	ELSE (* command not yet active *)
		IF F_AxisIsCoupled(Axis.NcToPlc.CoupleState) THEN	(* 20090205 KSt *)
			(* if axis is coupled during motion (FlyingSaw) all commands are aborted - 20090205 KSt*)
			CommandAborted := TRUE;
			iState := STATE_INITIALIZATION;
		ELSIF Axis.NcToPlc.CmdNo = 0 AND NcCyclicFeedbackExpected THEN  				(* 20090206 KSt *)
			CounterCmdNoZero := CounterCmdNoZero + 1;
			IF CounterCmdNoZero > TcMcGlobal.NCTOPLC_FEEDBACK_MAXWAITCYCLES THEN (* wait for a certain number of cycles before error *)
				(* CmdNo zero is not supposed to happen - it may come up after a coupling situation for a few cycles *)
				Error := TRUE;
				ErrorID := MC_ERROR_BUFFERED_COMMAND_CMDNOZERO; (* no command state feedback from NC *)
				iState := STATE_INITIALIZATION;
			END_IF
																														(*		ELSIF Axis.NcToPlc.CmdNo = (sStartResponse.nCmdNo + 1) OR
																																     	((Axis.NcToPlc.CmdNo = 1) AND  (sStartResponse.nCmdNo=16#FFFF)) *) 	(* overrun with a difference of 1*) 
		ELSIF DiffCmdNo=1 THEN (* running command number is 1 higher than expected *) (* 20110421 KSt *)
			(* feedback CmdNo is exactly ONE increment higher than my command *)
			(* command was aborted or successfully finished *)
			Error := GETBIT32(Axis.NcToPlc.CmdState, INT_TO_SINT(CMDSTATE_LASTCMD_ENDED_WITH_ERROR));
			CommandAborted := NOT Error AND GETBIT32(Axis.NcToPlc.CmdState, INT_TO_SINT(CMDSTATE_LASTCMD_ABORTED_WITHOUT_ERROR));
(*			Done := NOT Error AND NOT Done AND GETBIT32(Axis.NcToPlc.CmdState, INT_TO_SINT(CMDSTATE_LASTCMD_SUCCESSFULLY_EXECUTED));*)	(* 20100514 KSt *)
			Done := NOT Error AND NOT CommandAborted AND GETBIT32(Axis.NcToPlc.CmdState, INT_TO_SINT(CMDSTATE_LASTCMD_SUCCESSFULLY_EXECUTED));	(* 20100514 KSt *)
			IF Error THEN
				(* if axis error-Id is valid then feed it back - otherwhise errror-Id is unknown. *)
				ErrorID := SEL(Axis.NcToPlc.ErrorCode=0, Axis.NcToPlc.ErrorCode, INT_TO_UDINT(MC_ERROR_BUFFERED_COMMAND_ERRORID_NOT_AVAILABLE) );
			END_IF
			IF NOT Done AND NOT CommandAborted AND NOT Error THEN
				Error := TRUE;
				ErrorID := MC_ERROR_BUFFERED_COMMAND_NO_STATE_FEEDBACK; (* no command state feedback from NC *)
			END_IF
			iState := STATE_INITIALIZATION;
		ELSIF DiffCmdNo=2 THEN (* running command number is 2 higher than expected *) (* 20110421 KSt *)
			(* feedback CmdNo is exactly TWO increments higher than my command  - 20090116 KSt *)
			Error := GETBIT32(Axis.NcToPlc.CmdState, INT_TO_SINT(CMDSTATE_LASTCMD_ENDED_WITH_ERROR)); (* error of command+1 *)
			(* if command+1 was aborted then this command has been aborted as well *)
			CommandAborted := NOT Error AND GETBIT32(Axis.NcToPlc.CmdState, INT_TO_SINT(CMDSTATE_LASTCMD_ABORTED_WITHOUT_ERROR));
			IF NOT CommandAborted THEN
				(* if previous command has not been aborted - the status of this command is unknown *)
				Error := TRUE;	(* command monitoring not possible; probably because function block was not called cyclically *)
				ErrorID := SEL( DiffCycleCounter > 1, INT_TO_UDINT(MC_ERROR_BUFFERED_COMMAND_MONITORING_IMPOSSIBLE), INT_TO_UDINT(MC_ERROR_BUFFCMD_MONITRNGIMPOSS_FBNOTCALLEDCYC));	(* additional error code with command aborted - command monitoring impossible because the block is not called cyclically - 2011-08-01 KSt *)
			END_IF
			iState := STATE_INITIALIZATION;
		ELSIF DiffCmdNo > 0 THEN (* running command number is 3 or more higher than expected *) (* 20110421 KSt *)
			(* feedback CmdNo is THREE or more increments higher than my command *)
			(* command was aborted - command monitoring impossible *)
			Error := TRUE; 	(* command monitoring not possible; probably because function block was not called cyclically *)
			ErrorID := SEL( DiffCycleCounter > 1, INT_TO_UDINT(MC_ERROR_BUFFERED_COMMAND_MONITORING_IMPOSSIBLE), INT_TO_UDINT(MC_ERROR_BUFFCMD_MONITRNGIMPOSS_FBNOTCALLEDCYC)); (* additional error code with command aborted - command monitoring impossible because the block is not called cyclically - 2011-08-01 KSt *)
			(*CommandAborted := TRUE;*)	(*  20090116 KSt *)
			iState := STATE_INITIALIZATION;
		ELSIF F_AxisInErrorState(Axis.NcToPlc.StateDWord) THEN
			(* axis error came up before this command has been started *)
			Error := TRUE;
			ErrorID := AXIS.NcToPlc.ErrorCode;
			iState := STATE_INITIALIZATION;
		ELSIF NOT F_AxisHasJob(Axis.NcToPlc.StateDWord) AND NcCyclicFeedbackExpected THEN
			(* CmdNo is still lower than my command - command has not been initiated *)
			IF F_AxisHasBeenStopped(Axis.NcToPlc.StateDWord) THEN
				CommandAborted := TRUE;		(* stopp command aborts this command *)
				iState := STATE_INITIALIZATION;
			ELSE
				(* other cases are not supposed to happen and are error conditions *)
				CounterCmdNotStarted := CounterCmdNotStarted + 1;
				IF CounterCmdNotStarted > TcMcGlobal.NCTOPLC_FEEDBACK_MAXWAITCYCLES THEN (* wait for a certain number of cycles before error *)
					Error := TRUE;
					ErrorID := MC_ERROR_BUFFERED_COMMAND_NOT_STARTED; (* reason unknown *)
					iState := STATE_INITIALIZATION;
				END_IF
			END_IF
			(* timeout check *);
		END_IF
	END_IF
	IF (Error OR CommandAborted) AND (iState<>STATE_RUNNING) THEN
		ActErrorMessage();
	END_IF

ELSE  (* CASE : Unknown program state *)
	iState:= STATE_INITIALIZATION;
END_CASE

ADSbusy := fbAdsReadWrite.BUSY;
IF iState=STATE_INITIALIZATION THEN
	(* reset Busy immediately  when sequence ends *)
	IF Busy THEN
		LastExecutionResult.Done := Done;
		LastExecutionResult.CommandAborted := CommandAborted;
		LastExecutionResult.Error := Error;
		LastExecutionResult.ErrorID := ErrorID;
	END_IF
	Busy := FALSE;
	Active := FALSE;
END_IF
END_FUNCTION_BLOCK
ACTION ActCalcDiffCmdNo:
(* 20110421 KSt *)
(* calculate the difference between the responsed CmdNo and the actually running CmdNo *)
IF sStartResponse.nCmdNo = 0 OR Axis.NcToPlc.CmdNo = 0 THEN
	DiffCmdNo := -16#8000;	(* special invalid case - feedback is maximum negative difference *)
ELSIF sStartResponse.nCmdNo > 16#A000 AND Axis.NcToPlc.CmdNo < 16#4000 THEN
	(* overrun - running CmdNo is higher than the responded number *)
	DiffCmdNo := WORD_TO_INT(Axis.NcToPlc.CmdNo - sStartResponse.nCmdNo - 1);	(* substract -1 because 0 is an invalid command number *)
ELSIF sStartResponse.nCmdNo < 16#4000 AND Axis.NcToPlc.CmdNo > 16#A000 THEN
	(* overrun - running CmdNo is lower than the responded number *)
	DiffCmdNo := WORD_TO_INT(Axis.NcToPlc.CmdNo - sStartResponse.nCmdNo + 1);	(* add 1 because 0 is an invalid command number *)
ELSE
	DiffCmdNo := WORD_TO_INT(Axis.NcToPlc.CmdNo - sStartResponse.nCmdNo);
END_IF
END_ACTION
ACTION ActErrorMessage:
IF Axis.PlcToNc.ControlDWord.30 THEN (* bit 30 - debug mode enabled *)
	(* FEHLERMELDUNG *)
	sTempMsg	:= 'TCMC:UAS Axis '; 	(* UAS = universal axis start *)
	sTempMsg	:= CONCAT( sTempMsg, UDINT_TO_STRING( Axis.NcToPlc.AxisId ) );
	sTempMsg	:= CONCAT( sTempMsg, ', CmdNo: ' );
	sTempMsg	:= CONCAT( sTempMsg, UDINT_TO_STRING( sStartResponse.nCmdNo ) );
	IF Error THEN
		sTempMsg	:= CONCAT( sTempMsg, ', Error: 0x' );
		sTempMsg	:= CONCAT( sTempMsg, _F_TcMC_DWORD_TO_HEXSTR(ErrorID) );
	END_IF
	IF CommandAborted THEN
		sTempMsg	:= CONCAT( sTempMsg, ', ABORTED ' );
	END_IF
	sTempMsg	:= CONCAT( sTempMsg, ', StartType: ' );
	sTempMsg	:= CONCAT( sTempMsg, UDINT_TO_STRING( sStartRequest.nStartType ) );
	sTempMsg	:= CONCAT( sTempMsg, ', SetPos: ' );
	sTempMsg	:= CONCAT( sTempMsg, LREAL_TO_STRING( _F_TcMC_Round( Axis.NcToPlc.SetPos , 4) ) );
	sTempMsg	:= CONCAT( sTempMsg, ', SetVelo: ' );
	sTempMsg	:= CONCAT( sTempMsg, LREAL_TO_STRING( _F_TcMC_Round( Axis.NcToPlc.SetVelo, 4) ) );
	sTempMsg	:= CONCAT( sTempMsg, ', SetAcc: ' );
	sTempMsg	:= CONCAT( sTempMsg, LREAL_TO_STRING( _F_TcMC_Round( Axis.NcToPlc.SetAcc, 4) ) );
	sTempMsg	:= CONCAT( sTempMsg, ', PosTarget: ' );
	sTempMsg	:= CONCAT( sTempMsg, LREAL_TO_STRING( _F_TcMC_Round( sStartRequest.fPosTarget, 4) ) );
	sTempMsg	:= CONCAT( sTempMsg, ',  VeloRequ: ' );
	sTempMsg	:= CONCAT( sTempMsg, LREAL_TO_STRING( _F_TcMC_Round(sStartRequest.fVeloRequ, 4) ) );
	sTempMsg	:= CONCAT( sTempMsg, ',  Acc: ' );
	sTempMsg	:= CONCAT( sTempMsg, LREAL_TO_STRING( _F_TcMC_Round( sStartRequest.fAcc, 4) ) );
	sTempMsg	:= CONCAT( sTempMsg, ',  Dec: ' );
	sTempMsg	:= CONCAT( sTempMsg, LREAL_TO_STRING( _F_TcMC_Round( sStartRequest.fDec, 4) ) );
	sTempMsg	:= CONCAT( sTempMsg, ',  Jerk: ' );
	sTempMsg	:= CONCAT( sTempMsg, LREAL_TO_STRING( _F_TcMC_Round( sStartRequest.fJerk, 4) ) );
	sTempMsg	:= CONCAT( sTempMsg, ', BufMode: ' );
	sTempMsg	:= CONCAT( sTempMsg, UDINT_TO_STRING(sStartRequest.nBufferMode ) );
	sTempMsg	:= CONCAT( sTempMsg, ',  BlendPos: ' );
	sTempMsg	:= CONCAT( sTempMsg, LREAL_TO_STRING( _F_TcMC_Round( sStartRequest.fBlendingPosition, 4) ) );
	sTempMsg	:= CONCAT( sTempMsg, ',  ADS-Stamp: ' );
	sTempMsg	:= CONCAT( sTempMsg, UDINT_TO_STRING( fbAdsReadWrite.fbAdsRdWrt.STAMP_I) );

	(* additional PLC debug info for Beckhoff debugging programs *)
	(*
	IF Axis.PlcToNc.Reserved1 <> 0 THEN
		sTempMsg 	:= CONCAT( sTempMsg, ', PLC-Code=' );
		sTempMsg 	:= CONCAT( sTempMsg, DWORD_TO_STRING(PlcDebugCode) );
	END_IF
	*)
	IF Error THEN
		ADSLOGSTR( ADSLOG_MSGTYPE_ERROR + ADSLOG_MSGTYPE_LOG, sTempMsg, '' );		(* vom Typ <Fehlermeldung> *)
	ELSIF CommandAborted THEN
		ADSLOGSTR( ADSLOG_MSGTYPE_WARN, sTempMsg, '' ); 		(* vom Typ <Warnungsmeldung> *)
	ELSE
		ADSLOGSTR( ADSLOG_MSGTYPE_HINT, sTempMsg, '' ); 			(* vom Typ <Hinweismeldung> *)
	END_IF
END_IF
END_ACTION
ACTION ActMonitorContinousMotion:
(*
 * 	monitor continous motion
 *
 * 	monitor UNTIL the axis is in velocity AND the Execute-Input is FALSE
 * 	used with MoveVelocity and other continous commands
*)
IF F_AxisInErrorState(StateDWord := Axis.NcToPlc.StateDWord) THEN (* error while positioning *)
	Error := TRUE;
	ErrorID := Axis.NcToPlc.ErrorCode;
	InVelocity := FALSE;	(* reset InVelocity in case of error or abortion - KST 2012-05-16 *)
	iState := STATE_INITIALIZATION;
ELSIF NOT F_AxisHasJob(Axis.NcToPlc.StateDWord) OR F_AxisHasBeenStopped(Axis.NcToPlc.StateDWord) THEN (* KSt 27.5.03 *)
	(* aborted during accelertion *)
	CommandAborted := TRUE;
	InVelocity := FALSE;	(* reset InVelocity in case of error or abortion - KST 2012-05-16 *)
	iState := STATE_INITIALIZATION;
ELSIF InVelocity AND NOT Execute THEN
	(* end of axis control after beeing in velocity for at least one cycle *)
	iState := STATE_INITIALIZATION;
(* ELSIF Axis.NcToPlc.AxisState = TCNC_PHASE_VELOCONST THEN *)	(* 20100506 KST - changed for MoveContinous Absolute and MoveContinousRelative *)
(*ELSIF Axis.NcToPlc.AxisState = INT_TO_DWORD(TCNC_PHASE_VELOCONST) AND F_AxisIsMovingEndless(Axis.NcToPlc.StateDWord) THEN*)	(* 20100506 KST - changed for MoveContinous Absolute and MoveContinousRelative *)
ELSIF F_AxisIsMovingEndless(Axis.NcToPlc.StateDWord)	(* 20100506 KST - changed for MoveContinous Absolute and MoveContinousRelative *)
	AND ((Axis.NcToPlc.AxisState = INT_TO_DWORD(TCNC_PHASE_VELOCONST)) OR	(* continous axes *)
		   (Axis.NcToPlc.AxisState = INT_TO_DWORD(TCNC_PHASE_TWOSPEED_MOVING)) AND F_AxisReachedConstantVelocity(Axis.NcToPlc.StateDWord)) (* 20110719 KST - two speed axes *)
	THEN
	InVelocity := TRUE;
ELSIF InVelocity AND NOT F_AxisIsCompensating(Axis.NcToPlc.StateDWord) THEN
	(* axis was InVelocity but isn't any more, superposition is allowed but *)
	(* any other reason is an abortion *)
	CommandAborted := TRUE;
	InVelocity := FALSE;	(* reset InVelocity in case of error or abortion - KST 2012-05-16 *)
	iState := STATE_INITIALIZATION;
END_IF
Done := InVelocity;
END_ACTION
ACTION ActMonitorDiscreteMotion:
(*
 * 	monitor discrete motion 
 *
 *	monitor until the target position is reached 
 * 	used with MC_MoveAbsolute and other discrete commands
*)

(* check for reached target position *)
IF (Axis.NcToPlc.OpModeDWord AND  OpMode.TargetPosControl) > 0 THEN (* Target position controlling and PEH enabled ? *)
	IF NOT F_AxisHasJob(Axis.NcToPlc.StateDWord) AND F_AxisIsAtTargetPosition(Axis.NcToPlc.StateDWord) THEN
		Done := TRUE;
		iState := STATE_INITIALIZATION;
	END_IF
ELSE
	IF (Axis.NcToPlc.OpModeDWord AND OpMode.PosAreaControl) > 0 THEN (* Target position controlling enabled ? *)
		IF NOT F_AxisHasJob(Axis.NcToPlc.StateDWord) AND F_AxisInPositionWindow(Axis.NcToPlc.StateDWord) THEN
			Done := TRUE;
			iState := STATE_INITIALIZATION;
		END_IF
	ELSE
		IF NOT F_AxisHasJob(Axis.NcToPlc.StateDWord) THEN
			Done := TRUE;
			iState := STATE_INITIALIZATION;
		END_IF
	END_IF
END_IF;
(* check for timeout *)
IF NOT done AND NOT F_AxisHasJob(Axis.NcToPlc.StateDWord) THEN
	fbTimeOut(IN:= TRUE, PT:= TcMcGlobal.tTargetPosTimeOut);
	IF fbTimeOut.Q THEN
		Error := TRUE;
		ErrorID := MC_ERROR_TARGETPOS_TIMEOUT;
		iState := STATE_INITIALIZATION;
	END_IF;
END_IF;

(* error while positioning *)
IF	F_AxisInErrorState(Axis.NcToPlc.StateDWord) THEN
	Done := FALSE;	(* KSt - 2013-05-23 *)
	Error := TRUE;
	ErrorID := Axis.NcToPlc.ErrorCode;
	iState := STATE_INITIALIZATION;
ELSIF 	F_AxisHasBeenStopped(Axis.NcToPlc.StateDWord)
		AND NOT F_AxisHasJob(Axis.NcToPlc.StateDWord)
		AND NOT (StartType=TCNC_START_HALT)
		AND NOT (StartType=TCNC_START_STOPANDLOCK)
		THEN
		(* manual stop or stop FB ? *)
		Done := FALSE;	(* KSt - 2013-07-02 - reset Done in case of CommandAborted *)
(*		ErrorID := MC_ERROR_AXIS_HAS_BEEN_STOPPED;*)	(* HKP - 2013-07-02 - ErrorID removed because just informational feedback *)
		CommandAborted 	:= TRUE;
		iState := STATE_INITIALIZATION;
(*	bit 18 is not implemented - 20080610 KSt
ELSIF  F_AxisIsNotInTargetPosition(Axis.NcToPlc.StateDWord) THEN
	( target pos can NOT be reached )
		ErrorID := MC_ERROR_TARGETPOS_TIMEOUT;
		Error := TRUE;
		iState := STATE_INITIALIZATION;
*)
END_IF
END_ACTION
ACTION ActMonitorStop:
(*
 * 	monitor a motion stop or halt
 *
 *	monitor until the target position is reached 
 * 	used with MC_Halt and MC_Stop commands
*)

(* check for deceleration *)
fbTimeOut(IN:= Axis.NcToPlc.AxisState <> INT_TO_DWORD(TCNC_PHASE_ACCNEG) , PT:= TcMcGlobal.tTargetPosTimeOut);
fbStopMonitoringTimeOut();

(* error while positioning *)
IF	F_AxisInErrorState(Axis.NcToPlc.StateDWord) THEN
	Error := TRUE;
	ErrorID := Axis.NcToPlc.ErrorCode;
	iState := STATE_INITIALIZATION;

(* check for end of motion  *)
ELSIF NOT F_AxisHasJob(Axis.NcToPlc.StateDWord) THEN
	IF 	(Axis.NcToPlc.OpModeDWord AND OpMode.StopMonitoring) > 0 THEN	(* stop monitoring active *)
		(* 20111208 KSt - if stop monitoring is active, axis waits for actual position beeing in target window *)
		fbStopMonitoringTimeOut(IN:= TRUE, PT:= TcMcGlobal.tStopMonitoringTimeOut);	(* start monitoring timer *)
		IF F_AxisIsAtTargetPosition(Axis.NcToPlc.StateDWord) THEN
			(* axis is in standstill and the actual value is inside the monitoring window *)
			Done := TRUE;
			iState := STATE_INITIALIZATION;
		ELSIF  fbStopMonitoringTimeOut.Q THEN (* not error but end of monitoring *)
			(* axis set position is in standstill but the acutal value did probalby not reach the monitoring window - no error in this case *)
			Done := TRUE;
			iState := STATE_INITIALIZATION;
		END_IF
	ELSE
		(* done after has job false without other monitoring *)
		Done := TRUE;
		iState := STATE_INITIALIZATION;
	END_IF

(* check for timeout *)
ELSIF fbTimeOut.Q THEN
	Error := TRUE;
	ErrorID := MC_ERROR_TARGETPOS_TIMEOUT;
	iState := STATE_INITIALIZATION;
END_IF;
END_ACTION
ACTION ActNcCycleCounter:
(*
	check if cyclic NcToPlc interface changed.
	If not, any Error or CommandAborted condition will be delayed.
	This piece of code prevents from errors if the Plc is called faster than the NC.
	2009-12-08 KSt
*)

fbTimeOutMappingCounter( IN := NcMappingCounter=0, PT:= t#50ms );	(* timout if no nc cyclic feedback for a while *)

NcCycleCounter := DWORD_TO_BYTE(SHR(Axis.NcToPlc.OpModeDWord, 24));
IF NcCycleCounter <> LastNcCycleCounter THEN
	NcMappingCounter := NcMappingCounter + 1; (* has been reset when the command was initiated *)
	NcCycleCounterAvailable := TRUE; (* marked as available when first time not zero - this flag will never be reset at run-time *)
	NcCycleCounterNotAvailable := FALSE;
ELSIF NOT NcCycleCounterAvailable AND fbTimeOutMappingCounter.Q THEN
	NcCycleCounterNotAvailable := TRUE; (* not available on old target systems *)
END_IF
LastNcCycleCounter:=NcCycleCounter;

IF NcCycleCounterNotAvailable OR (NcMappingCounter > 1) OR fbTimeOutMappingCounter.Q THEN
	(*	NcMappingCounter is set to TRUE after an ADS command has been answered.
		NcCyclicFeedbackExpected is set to TRUE when the NcMappingCounter has been 
		incremented at least twice after an ADS command.
		Also TRUE when cycle counter is not available on old target systems and after a time-out 
	*)
	(* 	If NcCyclicFeedbackExpected is false any wrong condition detected from the
		cyclic NcToPlc interface cannot lead to an Error or CommandAborted result.
	*)
	NcCyclicFeedbackExpected := TRUE;
END_IF
END_ACTION

(* POU F_AxisInProtectedMode, ST *)
FUNCTION F_AxisInProtectedMode  : BOOL
(* 	reference: 	NC -> PLC axis interface (128 bytes)
	check if bit 5 of an axis StateDWord is set:
	Axis is in a protected operating mode (e.g. as a slave axis, or under axis interpolation)
	Achse ist in geschützter Betriebsart (z.B. Slave-Achse oder Achsinterpolation)
*)
VAR_INPUT
	StateDWord : DWORD;
END_VAR
VAR
END_VAR
F_AxisInProtectedMode := (StateDWord AND 2#0000_0000_0000_0000_0000_0000_0010_0000) <> 0;
END_FUNCTION

(* POU F_AxisHasExtSetPointGen, ST *)
FUNCTION F_AxisHasExtSetPointGen : BOOL
(* 	reference: 	NC -> PLC axis interface (128 bytes)
	check if bit 14 of an axis StateDWord is set:
	Axis has an external set point generator (PLC)
	Achse hat einen externen Sollwertgenerator (SPS)
*)
VAR_INPUT
	StateDWord : DWORD;
END_VAR
VAR
END_VAR
F_AxisHasExtSetPointGen := (StateDWord AND 2#0000_0000_0000_0000_0100_0000_0000_0000) <> 0;
END_FUNCTION

(* POU F_AxisReachedConstantVelocity, ST *)
FUNCTION F_AxisReachedConstantVelocity  : BOOL
(* 	reference: 	NC -> PLC axis interface (128 bytes)
	check if bit 12 of an axis StateDWord is set:
	Axis has reached its constant velocity or rotary speed
	Achse hat V-Konst bzw. Drehzahl erreicht
*)
VAR_INPUT
	StateDWord : DWORD;
END_VAR
VAR
END_VAR
F_AxisReachedConstantVelocity := (StateDWord AND 2#0000_0000_0000_0000_0001_0000_0000_0000) <> 0;
END_FUNCTION

(* POU F_AxisIsCompensating, ST *)
FUNCTION F_AxisIsCompensating  : BOOL
(* 	reference: 	NC -> PLC axis interface (128 bytes)
	check if bit 13 of an axis StateDWord is set:
 	After a "Distance Compensation" is startet this bit means:
	Axis is in compensation mode
*)
VAR_INPUT
	StateDWord : DWORD;
END_VAR
VAR
END_VAR
F_AxisIsCompensating := (StateDWord AND 2#0000_0000_0000_0000_0010_0000_0000_0000) <> 0;
END_FUNCTION

(* POU MC_MoveAbsolute, FBD *)
FUNCTION_BLOCK MC_MoveAbsolute
(*	This Function Block commands a controlled motion to a specified absolute position.	*)
VAR_IN_OUT
	Axis				:	AXIS_REF;	(* B *)
END_VAR
VAR_INPUT
	Execute			:	BOOL;	(* B *)	(* Start the motion at rising edge *)
(*	ContinuousUpdate :	BOOL; *)	(* E *)	(* not available *)
	Position			:	LREAL;	(* B *)	(* Target position for the motion *)
	Velocity			:	LREAL;	(* E *)	(* Value of the maximum velocity *)
	Acceleration		:	LREAL;	(* E *)	(* Value of the maximum acceleration *)
	Deceleration		:	LREAL;	(* E *)	(* Value of the maximum deceleration *)
	Jerk				:	LREAL;	(* E *)	(* Value of the maximum jerk *)
(*	Direction			:	MC_Direction; *)	(* E *)	(* not available *)
	BufferMode		:	MC_BufferMode;	(* E *)
	Options			: 	ST_MoveOptions;	(* V *)	(* optional parameters *)
END_VAR
VAR_OUTPUT
	Done			:	BOOL;	(* B *)
	Busy			: 	BOOL;	(* E *)
	Active			: 	BOOL;	(* E *)
	CommandAborted	:	BOOL;	(* E *)
	Error			:	BOOL;	(* B *)
	ErrorID			:	UDINT;	(* E *)
END_VAR
VAR
	LastExecutionResult: 	_ST_FunctionBlockResults;
	ADSbusy		: 	BOOL;
	MoveGeneric		: 	_FB_MoveUniversalGeneric;
	CmdNo: UINT;
END_VAR
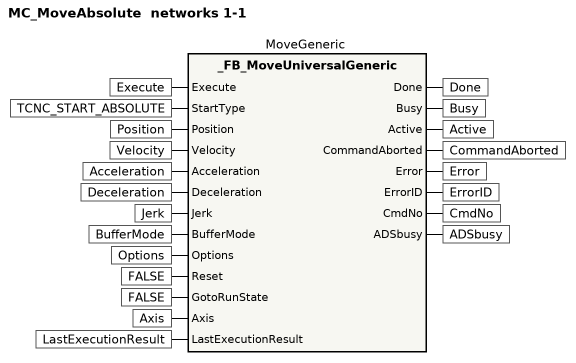
_FBD_ (* Function Block Diagram *)
NETWORK 1 (* PlcOpen comment / The >ContinousUpdate< input is not supported / The >Direction< input is not supported *)
	MoveGeneric :_FB_MoveUniversalGeneric(Execute: Execute, StartType: TCNC_START_ABSOLUTE, Position: Position, Velocity: Velocity, Acceleration: Acceleration, Deceleration: Deceleration, Jerk: Jerk, BufferMode: BufferMode, Options: Options, Reset: FALSE, GotoRunState: FALSE, Axis: Axis, LastExecutionResult: LastExecutionResult, Busy => Busy, Active => Active, CommandAborted => CommandAborted, Error => Error, ErrorID => ErrorID, CmdNo => CmdNo, ADSbusy => ADSbusy) => Done
_END_FBD_
(* the same logic as Structured Text *)
(* Network 1: PlcOpen comment / The >ContinousUpdate< input is not supported / The >Direction< input is not supported *)
MoveGeneric (Execute := Execute, StartType := TCNC_START_ABSOLUTE, Position := Position, Velocity := Velocity, Acceleration := Acceleration, Deceleration := Deceleration, Jerk := Jerk, BufferMode := BufferMode, Options := Options, Reset := FALSE, GotoRunState := FALSE, Axis := Axis, LastExecutionResult := LastExecutionResult);
Busy := MoveGeneric .Busy;
Active := MoveGeneric .Active;
CommandAborted := MoveGeneric .CommandAborted;
Error := MoveGeneric .Error;
ErrorID := MoveGeneric .ErrorID;
CmdNo := MoveGeneric .CmdNo;
ADSbusy := MoveGeneric .ADSbusy;
Done := MoveGeneric .Done;
END_FUNCTION_BLOCK

(* POU F_AxisIsAtTargetPosition, ST *)
FUNCTION F_AxisIsAtTargetPosition  : BOOL
(* 	reference: 	NC -> PLC axis interface (128 bytes)
	check if bit 4 of an axis StateDWord is set:
	Axis is at target position (PEH) (physical feedback)
	Achse ist in Zielposition (PEH) (physik. Rückmeldung)
*)
VAR_INPUT
	StateDWord : DWORD;
END_VAR
VAR
END_VAR
F_AxisIsAtTargetPosition := (StateDWord AND 2#0000_0000_0000_0000_0000_0000_0001_0000) <> 0;
END_FUNCTION

(* POU F_AxisInPositionWindow, ST *)
FUNCTION F_AxisInPositionWindow : BOOL
(* 	reference: 	NC -> PLC axis interface (128 bytes)
	check if bit 3 of an axis StateDWord is set:
	Axis is in position window (physical feedback)
	Achse ist im Positionsbereichsfenster (physik. Rückmeldung) 
*)
VAR_INPUT
	StateDWord : DWORD;
END_VAR
VAR
END_VAR
F_AxisInPositionWindow := (StateDWord AND 2#0000_0000_0000_0000_0000_0000_0000_1000) <> 0;
END_FUNCTION

(* POU MC_Halt, FBD *)
FUNCTION_BLOCK MC_Halt
(*	This function block commands a controlled motion stop. The axis is moved to
	the state 'DiscreteMotion', until the velocity is zero. With the Done output set, the 
	state is transferred to StandStill.

	Notes:
	- MC_Halt is used to stop the axis under normal operation conditions. 
	  In non-buffered mode it is possible to set another motion command during 
	  deceleration of the axis, which will abort the MC_Halt and will be executed 
	  immediately.
	- If this command is active the next command can be issued. 
	  E.g. a driverless vehicle detects an obstacle and needs to stop. 
	  MC_Halt is issued. Before the standstill is reached the obstacle is 
	  removed and the motion can be continued by setting another motion 
	  command, so the vehicle does not stop.
*)
VAR_IN_OUT
	Axis				:	AXIS_REF;	(* B *)
END_VAR
VAR_INPUT
	Execute			:	BOOL;	(* B *)
	Deceleration		:	LREAL;	(* E *)
	Jerk				:	LREAL;	(* E *)
	BufferMode		:	MC_BufferMode;	(* E *)
	Options			: 	ST_MoveOptions;	(* V *) (* optional parameters *)
END_VAR
VAR_OUTPUT
	Done			:	BOOL;	(* B *)
	Busy			: 	BOOL;	(* E *)
	Active			: 	BOOL;	(* E *)
	CommandAborted	:	BOOL;	(* E *)
	Error			:	BOOL;	(* B *)
	ErrorID			:	UDINT;	(* E *)
END_VAR
VAR
	LastExecutionResult: 	_ST_FunctionBlockResults;
	ADSbusy		: 	BOOL;
	MoveGeneric		: 	_FB_MoveUniversalGeneric;
	CmdNo: UINT;
END_VAR
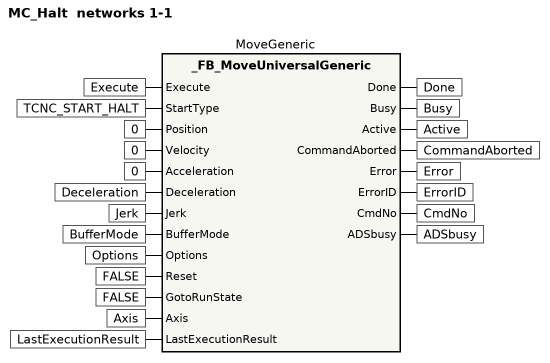
_FBD_ (* Function Block Diagram *)
NETWORK 1
	MoveGeneric   :_FB_MoveUniversalGeneric(Execute: Execute, StartType: TCNC_START_HALT, Position: 0, Velocity: 0, Acceleration: 0, Deceleration: Deceleration, Jerk: Jerk, BufferMode: BufferMode, Options: Options, Reset: FALSE, GotoRunState: FALSE, Axis: Axis, LastExecutionResult: LastExecutionResult, Busy => Busy, Active => Active, CommandAborted => CommandAborted, Error => Error, ErrorID => ErrorID, CmdNo => CmdNo, ADSbusy => ADSbusy) => Done
_END_FBD_
(* the same logic as Structured Text *)
(* Network 1 *)
MoveGeneric   (Execute := Execute, StartType := TCNC_START_HALT, Position := 0, Velocity := 0, Acceleration := 0, Deceleration := Deceleration, Jerk := Jerk, BufferMode := BufferMode, Options := Options, Reset := FALSE, GotoRunState := FALSE, Axis := Axis, LastExecutionResult := LastExecutionResult);
Busy := MoveGeneric   .Busy;
Active := MoveGeneric   .Active;
CommandAborted := MoveGeneric   .CommandAborted;
Error := MoveGeneric   .Error;
ErrorID := MoveGeneric   .ErrorID;
CmdNo := MoveGeneric   .CmdNo;
ADSbusy := MoveGeneric   .ADSbusy;
Done := MoveGeneric   .Done;
END_FUNCTION_BLOCK

(* POU MC_Stop, ST *)
FUNCTION_BLOCK MC_Stop
(*	This FB is primarily intended for emergency stop functionality or exception
	situations.
	This Function Block commands a controlled motion stop and transfers the
	axis to the state 'Stopping'. While the axis is in state Stopping, no other FB 
	can perform any motion on the same axis. After the axis has reached velocity 
	zero, the Done output is set to TRUE immediately. The axis remains in the 
	state 'Stopping' as long as Execute is still TRUE or velocity zero is not yet 
	reached. As soon as 'Done' is set and 'Execute' is FALSE the axis goes to 
	state 'StandStill'.
*)
VAR_IN_OUT
	Axis				:	AXIS_REF;	(* B *)
END_VAR
VAR_INPUT
	Execute			:	BOOL;	(* B *)
	Deceleration		:	LREAL;	(* E *)
	Jerk				:	LREAL;	(* E *)
(*	BufferMode		:	MC_BufferMode;*)	(* E *) (* 2008-06-27 KSt - deleted after PlcOpen corrigendum V0.4 *)
	Options			: 	ST_MoveOptions;	(* V *) (* optional parameters *)
END_VAR
VAR_OUTPUT
	Done			:	BOOL;	(* B *)
	Busy			: 	BOOL;	(* E *)
	Active			: 	BOOL;	(* E *)
	CommandAborted	:	BOOL;	(* E *)
	Error			:	BOOL;	(* B *)
	ErrorID			:	UDINT;	(* E *)
END_VAR
VAR
	LastExecutionResult: 	_ST_FunctionBlockResults;
	ADSbusy		: 	BOOL;
	MoveGeneric		: 	_FB_MoveUniversalGeneric;
	ReleaseLock		: 	ADSWRITE;
	CmdNo			: 	UINT;
	AxisMotionCommandsLocked		: 	BOOL;
	iState			: 	_E_TcMC_STATES := STATE_INITIALIZATION;
	NoJobTimer		: 	TON;
END_VAR
{library private}
VAR
	fbOnTrigger		: 	R_TRIG;
	CounterMotionCommandsLocked: INT;
END_VAR
fbOnTrigger(CLK:= Execute);

CASE iState OF
STATE_INITIALIZATION:	(* *)
	Busy := FALSE;
	Active := FALSE;
	IF NOT Execute THEN
		Done := FALSE;
		CommandAborted := FALSE;
		Error := FALSE;			(* reset at falling edge of Execute *)
		ErrorID := 0;
	END_IF
    	IF fbOnTrigger.Q THEN
		(* initialize output values *)
		Done := FALSE;
		Busy := TRUE;
		Active := FALSE;
		CommandAborted := FALSE;
		Error := FALSE;
		ErrorID := 0;
		ReleaseLock.WRITE:=FALSE;
		NoJobTimer( IN:=FALSE);	(* 20111209 KSt *)
		iState := STATE_ORDER;
	END_IF

STATE_ORDER :
	(* wait until stop is getting active or axis has stopped for a reason *)
	IF 	MoveGeneric.Active OR
		NOT F_AxisHasJob(Axis.NcToPlc.StateDWord)
		THEN
		Active := TRUE;
		ActStop();
		IF NOT ReleaseLock.BUSY THEN (* may be busy after fast stop retrigger *)
			ReleaseLock.WRITE:=FALSE;
			CounterMotionCommandsLocked := 0;
			iState := STATE_RUNNING;
		END_IF
	ELSIF MoveGeneric.Error OR MoveGeneric.CommandAborted THEN	(* ELSIF added 2009-11-09 KSt *)
		Error := MoveGeneric.Error;
		ErrorID := MoveGeneric.ErrorID;
		CommandAborted := MoveGeneric.CommandAborted;
		IF F_AxisHasJob(Axis.NcToPlc.StateDWord) AND NOT F_AxisMotionCommandsLocked(Axis.NcToPlc.StateDWord) THEN
			iState := STATE_INITIALIZATION; (* command not accepted *)
		ELSIF Execute THEN
			iState := STATE_MOTIONCOMMANDSLOCKED;	(* wait to release after Execute is FALSE *)
		ELSE
			ReleaseLock.WRITE := TRUE;	(* release axis if Execute is already FALSE *)
			iState := STATE_WAITING;
		END_IF
	END_IF

STATE_RUNNING:  (* wait until axis stands still and Execute is FALSE *)
	(* axis is stopping during this state *)
	IF NOT F_AxisHasJob(Axis.NcToPlc.StateDWord) THEN
		NoJobTimer.IN := TRUE;
	END_IF
	NoJobTimer( PT:=TcMcGlobal.tStopMonitoringTimeOut + T#50ms );	(* 20111209 KSt - just a safety timer - typically not relevant if MoveGeneric is working correctly *)
	IF 	NOT MoveGeneric.Busy OR					(* successfully stopped *)
		(* NOT F_AxisHasJob(Axis.NcToPlc.StateDWord)*) (* or in standstill for any other reason *)	(* 20111209 KSt *)
		NoJobTimer.Q (* or in standstill for any other reason *)	(* 20111209 KSt *)
		THEN
		Error := MoveGeneric.Error;		(* 2008-11-26 KSt *)
		ErrorID := MoveGeneric.ErrorID;	(* 2008-11-26 KSt *)
		CommandAborted := MoveGeneric.CommandAborted;	(* KSt 2009-04-15 *)
		Done := NOT Error AND NOT CommandAborted;		(* KSt 2009-04-15 *)
		IF Execute THEN
			iState := STATE_MOTIONCOMMANDSLOCKED;
		ELSE
			ReleaseLock.WRITE := TRUE;	(* release axis if Execute is already FALSE *)
			iState := STATE_WAITING;
		END_IF
	END_IF

STATE_MOTIONCOMMANDSLOCKED : 	(* axis is in standstill and axis is locked against motion commands during this state *)
	IF AxisMotionCommandsLocked AND NOT F_AxisMotionCommandsLocked(Axis.NcToPlc.StateDWord) THEN (* IF block added 2015-03-19 KSt *)
		(* if axis was locked but is not locked anymore it may have been released by a axis reset command *)
		(* IF block added 2015-03-19 KSt *)
		Done := FALSE;
		CommandAborted := NOT Error;
		iState := STATE_INITIALIZATION;
	ELSIF NOT Execute THEN	(* reset outputs if Execute is FALSE *)
		Done := FALSE;
		CommandAborted := FALSE;
		Error := FALSE;
		ErrorID := 0;
		ReleaseLock.WRITE:=TRUE;	(* release axis *)
		CounterMotionCommandsLocked := 0;
		iState := STATE_WAITING;
	END_IF

STATE_WAITING : (* release axis and wait until axis is released *)
	IF NOT Execute THEN	(* reset outputs if Execute is FALSE *)
		Done := FALSE;
		CommandAborted := FALSE;
		Error := FALSE;
		ErrorID := 0;
	END_IF
	ReleaseLock.WRITE:=TRUE;
	ActStop(); (* call here - fast reaction required *)
	IF NOT ReleaseLock.BUSY THEN
		IF ReleaseLock.ERR THEN
			Error := TRUE;
			ErrorID := ReleaseLock.ERRID;
			iState := STATE_INITIALIZATION;
		(* ELSIF NOT F_AxisMotionCommandsLocked(Axis.NcToPlc.StateDWord) THEN *) (* NOT deleted 2009-05-11 KSt *)
		ELSIF F_AxisMotionCommandsLocked(Axis.NcToPlc.StateDWord) THEN
			CounterMotionCommandsLocked := CounterMotionCommandsLocked + 1; (* wait for a certain number of cycles before error - 2009-10-06 KSt *)
			IF CounterMotionCommandsLocked > TcMcGlobal.NCTOPLC_FEEDBACK_MAXWAITCYCLES THEN
				Error := TRUE;
				ErrorID := MC_ERROR_BUFFERED_COMMAND_NO_STATE_FEEDBACK; (* lock bit has not been reset *)
				iState := STATE_INITIALIZATION;
			END_IF
		ELSE (* axis released - no error *)
			iState := STATE_INITIALIZATION;
		END_IF
		ReleaseLock.WRITE:=FALSE;
	END_IF

    	IF fbOnTrigger.Q THEN (* KSt 2009-04-15 - Stop retrigger allowed after release even without a "released" feedback*)
		(* initialize output values *)
		Done := FALSE;
		Busy := TRUE;
		Active := FALSE;
		CommandAborted := FALSE;
		Error := FALSE;
		ErrorID := 0;
		ReleaseLock.WRITE:=FALSE;
		iState := STATE_ORDER;	(* retrigger stop command *)
	END_IF

END_CASE

ActStop(); (* call function blocks *)

ADSbusy := MoveGeneric.ADSbusy OR ReleaseLock.BUSY;
IF iState=STATE_INITIALIZATION THEN
	(* reset Busy immediately  when sequence ends *)
	Done:=FALSE;
	Busy := FALSE;
	Active := FALSE;
END_IF
END_FUNCTION_BLOCK
ACTION ActStop:
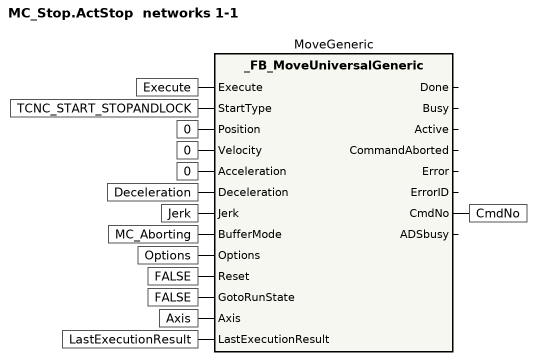
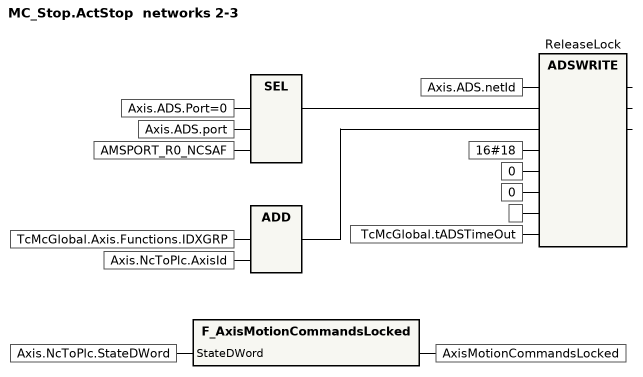
_FBD_ (* Function Block Diagram *)
NETWORK 1
	MoveGeneric:_FB_MoveUniversalGeneric(Execute: Execute, StartType: TCNC_START_STOPANDLOCK, Position: 0, Velocity: 0, Acceleration: 0, Deceleration: Deceleration, Jerk: Jerk, BufferMode: MC_Aborting, Options: Options, Reset: FALSE, GotoRunState: FALSE, Axis: Axis, LastExecutionResult: LastExecutionResult, CmdNo => CmdNo)
NETWORK 2 (* Release locked axis after it has been locked by the MC_Stop command *)
	ReleaseLock:ADSWRITE(Axis.ADS.netId, SEL(Axis.ADS.Port=0, Axis.ADS.port, AMSPORT_R0_NCSAF), ADD(TcMcGlobal.Axis.Functions.IDXGRP, Axis.NcToPlc.AxisId), 16#18, 0, 0, ,  TcMcGlobal.tADSTimeOut)
NETWORK 3
	F_AxisMotionCommandsLocked(StateDWord: Axis.NcToPlc.StateDWord) => AxisMotionCommandsLocked
_END_FBD_
(* the same logic as Structured Text *)
(* Network 1 *)
MoveGeneric(Execute := Execute, StartType := TCNC_START_STOPANDLOCK, Position := 0, Velocity := 0, Acceleration := 0, Deceleration := Deceleration, Jerk := Jerk, BufferMode := MC_Aborting, Options := Options, Reset := FALSE, GotoRunState := FALSE, Axis := Axis, LastExecutionResult := LastExecutionResult);
CmdNo := MoveGeneric.CmdNo;
(* Network 2: see the listing above *)
(* Network 3 *)
AxisMotionCommandsLocked := F_AxisMotionCommandsLocked(StateDWord := Axis.NcToPlc.StateDWord);
END_ACTION

(* POU _FB_PhasingGeneric, ST *)
FUNCTION_BLOCK _FB_PhasingGeneric
VAR_IN_OUT
	Master 			: 	AXIS_REF;
	Slave 			: 	AXIS_REF;
END_VAR
VAR_INPUT
	Execute			:	BOOL;	(* B *)	(* Start the motion at rising edge *)
(*	StartType		: 	UDINT;*)			(* command type start, stop etc, *)
	StartType		: 	_E_TcNC_StartPosType;	(* command type start, stop etc, *) (* 20110511 KSt type adaption for TC3 *)
	PhaseShift		:	LREAL;	(* B *)	(* Target position for the motion *)
	PhasingType		: 	E_PhasingType;	(* type of phase shift value, absolute or relative *)
	Velocity			:	LREAL;	(* E *)	(* Value of the maximum velocity *)
	Acceleration		:	LREAL;	(* E *)	(* Value of the maximum acceleration *)
	Deceleration		:	LREAL;	(* E *)	(* Value of the maximum deceleration *)
	Jerk				:	LREAL;	(* E *)	(* Value of the maximum jerk *)
	BufferMode		:	MC_BufferMode;		(* E *)
	Options			: 	ST_PhasingOptions;	(* V *)	(* optional parameters *)
END_VAR
VAR_OUTPUT
	Done			:	BOOL;	(* B *)
	Busy			: 	BOOL;	(* E *)
	Active			: 	BOOL;	(* E *)
	CommandAborted	:	BOOL;	(* E *)
	Error			:	BOOL;	(* B *)
	ErrorID			:	UDINT;	(* E *)
	PhaseShiftFeedback : 	LREAL;	(* E *)
END_VAR
VAR
	LastExecutionResult: 	_ST_FunctionBlockResults;
	ADSbusy		: 	BOOL;
	iState			:	_E_TcMC_STATES := STATE_INITIALIZATION;
(*	fbAdsReadWrite	: 	ADSRDWRTEX;*)
	fbAdsWrite		: 	ADSWRITE;
	sNcPhasing		: 	_ST_TcNC_PhasingRequest;
	PhasingStarted: BOOL;
END_VAR
{library private}
VAR
	fbTrigger			:	R_TRIG;
	fbTimeOut		: 	TON;
END_VAR
(* ====================================================================== *)
(* *)
(* ====================================================================== *)
fbTrigger(CLK:= Execute);

CASE iState OF
STATE_INITIALIZATION:	(* *)
	Busy := FALSE;
	Active := FALSE;

	IF NOT Execute THEN
		Done := FALSE;
		CommandAborted := FALSE;
		Error := FALSE;			(* reset at falling edge of Execute *)
		ErrorID := 0;
	END_IF;

    	IF fbTrigger.Q THEN
		(* initialize output values *)
		Done := FALSE;
		Busy := TRUE;
		CommandAborted := FALSE;
		Error := FALSE;
		ErrorID := 0;
		LastExecutionResult.Done := FALSE;
		LastExecutionResult.CommandAborted := FALSE;
		LastExecutionResult.Error := FALSE;
		LastExecutionResult.ErrorID := 0;
		PhaseShiftFeedback := 0;
		fbTimeOut(IN:= FALSE);
		fbAdsWrite(WRITE:=FALSE);

		(* fill structure *)
		sNcPhasing.nPhasingType	:= PhasingType;
		sNcPhasing.nControlMask 	:= 0;				(* not yet implemented *)
		sNcPhasing.fPhaseShift	:= PhaseShift;
		sNcPhasing.fVelo			:= Velocity;
		sNcPhasing.fAcc			:= Acceleration;
		sNcPhasing.fDec			:= Deceleration;
		sNcPhasing.fJerk			:= Jerk;
		sNcPhasing.nMasterAxisID	:= Master.NcToPlc.AxisId;
		sNcPhasing.nBufferMode	:= BufferMode;	(* not yet implemented *)
		sNcPhasing.fBlendingPos	:= 0;				(* not yet implemented *)

		fbAdsWrite.PORT := SEL(Slave.ADS.Port = 0, Slave.ADS.port, AMSPORT_R0_NCSAF);	(* KSt, 20090123 *)
		fbAdsWrite(	NETID:= TcMcGlobal.NCNETID_TCMC,
					IDXGRP:= TcMcGlobal.Axis.Functions.IDXGRP+Slave.NcToPlc.AxisId,
					IDXOFFS:= TcMcGlobal.Axis.Functions.IDXOFFS.PHASINGREQEUST,
					LEN:= SIZEOF(sNcPhasing),
					SRCADDR:= ADR(sNcPhasing),
					WRITE:= TRUE,
					TMOUT:= TcMcGlobal.tADSTimeOut );

		iState := STATE_ORDER;
	END_IF;

STATE_ORDER:  (* wait until command is accepted *)
	fbAdsWrite(WRITE:= TRUE);
	IF NOT fbAdsWrite.Busy THEN
		IF fbAdsWrite.Err THEN
			Error := TRUE;
			ErrorID := fbAdsWrite.ErrId;
			iState := STATE_INITIALIZATION;
		ELSE
			PhaseShiftFeedback := sNcPhasing.fPhaseShift;
			Active := TRUE;
			PhasingStarted := F_AxisPhasingActive(Slave.NcToPlc.StateDWord) ;
			iState := STATE_RUNNING;
		END_IF;
	END_IF;

STATE_RUNNING:  (* wait until axis stands still *)
	IF F_AxisPhasingActive(Slave.NcToPlc.StateDWord) THEN 	(* KSt, 29.4.2008 *)
		PhasingStarted := TRUE;
	ELSIF PhasingStarted  OR (StartType=TCNC_START_STOPANDLOCK) (* AND phasing  finished now *) THEN
		Done := TRUE;
		iState := STATE_INITIALIZATION;
	ELSE (* phasing operation did not start so far *)
		(* check for superposition not beeing started (KSt, 12.01.2004) *)
		fbTimeOut(IN:= TRUE, PT:= T#50ms);
		IF fbTimeOut.Q THEN
			(*	when the ADS command comes back without any error but
				the phasing operation does not start anyway, we assume that  
				a very short phasing operation has already been executed. 
			*)
			Done := TRUE; (* after short timeout *)
			iState := STATE_INITIALIZATION;
		END_IF;
	END_IF

ELSE  (* CASE : Unknown program state *)
	Error := TRUE;
	ErrorID := 16#FFFFFFFF;
	iState:= STATE_INITIALIZATION;
END_CASE

ADSbusy := fbAdsWrite.BUSY;
IF iState=STATE_INITIALIZATION THEN
	(* reset Busy immediately  when sequence ends *)
	IF Busy THEN
		LastExecutionResult.Done := Done;
		LastExecutionResult.CommandAborted := CommandAborted;
		LastExecutionResult.Error := Error;
		LastExecutionResult.ErrorID := ErrorID;
	END_IF
	Busy := FALSE;
	Active := FALSE;
END_IF
END_FUNCTION_BLOCK

(* POU F_AxisPhasingActive, ST *)
FUNCTION F_AxisPhasingActive  : BOOL
(* 	reference: 	NC -> PLC axis interface (128 bytes)
	check if bit 15 of an axis StateDWord is set:
	This bit is set while a phasing operation is busy.
	The flag is used at a slave axis of a coupling.
*)
VAR_INPUT
	StateDWord : DWORD;
END_VAR
VAR
END_VAR
F_AxisPhasingActive := (StateDWord AND 2#0000_0000_0000_0000_1000_0000_0000_0000) <> 0;
END_FUNCTION

(* POU _FB_PositionCorrectionTableLookup, ST *)
(*==========================================================================*)
(* Name:	_FB_PositionCorrectionTableLookup (based on FB_PositionCompensation)	*)
(* Parameter:	returns a compensation value depending on the position of the reference	*)
(*			axis																*)
(*																			*)
(* Author:	 	kbn & HKP														*)
(* Date:		06-July-2012														*)
(* last edit:	VER 2.0.0														*)
(*==========================================================================*)
FUNCTION_BLOCK _FB_PositionCorrectionTableLookup
VAR_IN_OUT
	Axis				: Axis_Ref;
END_VAR
VAR_INPUT
	Enable			: BOOL; 				(* rising edge triggers initialize routine *)
	pTable			: POINTER TO ST_PositionCompensationTableElement;	(* pointer to table of this type *)
	TableSize		: UDINT;				(* size of data in bytes related to 'pTable' *)
	TableParameter	: ST_PositionCompensationTableParameter;	(* position compensation table parameter structure *)
END_VAR
VAR_OUTPUT
	Compensation	: LREAL;
	Error			: BOOL;
	ErrorID			: UDINT;
	Active			: BOOL;
END_VAR
VAR
	nState			: UDINT;
	dwSize			: DWORD;
	eActiveDirection	: E_WorkDirection := WorkDirectionNone;
	bExecCalc		: BOOL;
	stElement1		: ST_PositionCompensationTableElement;
	stElement2		: ST_PositionCompensationTableElement;
	nLeftIndex		: UDINT;									(* Index starting from 0 up to (N-1) *)
	fSetPos			: LREAL;									(* position setpoint (absolute linear position or modulo position) *)
	(* HKP *)
	pTmpTable		: POINTER TO ST_PositionCompensationTableElement;	(* helper variable: pointer to table of this type *)
	fTmpStep		: LREAL;									(* helper variable *)
	fTmpA			: LREAL;									(* helper variable *)
	fTmpB			: LREAL;									(* helper variable *)
	fTmpDelta1		: LREAL;									(* helper variable *)
	fTmpDelta2		: LREAL;									(* helper variable *)
END_VAR
VAR CONSTANT
	ERRORCODE_PARAMSIZE	: UDINT := 16#4B43;
	ERRORCODE_PARAMPOS	: UDINT := 16#4B44;
(*	ERRORCODE_TCNCNOTIMPL	: UDINT := 16#4B45; *)
END_VAR
(* get last commanded direction *)
IF Axis.NcToPlc.SetVelo > 0.0001 THEN
	eActiveDirection	:= WorkDirectionPositive;
ELSIF Axis.NcToPlc.SetVelo < -0.0001 THEN
	eActiveDirection	:= WorkDirectionNegative;
END_IF

CASE nState OF
0:
	Error			:= FALSE;
	ErrorId			:= 0;
	Compensation	:= 0.0;
	Active			:= FALSE;
	bExecCalc		:= FALSE;

	IF Enable THEN
		(* reinitialize *)
		IF ( ABS(Axis.NcToPlc.SetVelo) < 0.0001 ) THEN
			eActiveDirection := WorkDirectionNone;
		END_IF
		(* check table size (in mimimum 2 elements needed) *)
		IF TableParameter.NoOfTableElements < 2 THEN
			Error	:= TRUE;
			ErrorId	:= ERRORCODE_PARAMSIZE;
			nState	:= 9999;
			RETURN;
		END_IF
		(* check table size *)
		IF TableParameter.NoOfTableElements*SIZEOF(pTable^) <> TableSize THEN
			Error	:= TRUE;
			ErrorId	:= ERRORCODE_PARAMSIZE;
			nState	:= 9999;
			RETURN;
		END_IF
		(* ====================================================== *)
		(* HKP: read table element with index (0)						*)
		(* ====================================================== *)
		(* stElement1	:= F_GetCompensationElementAt(pTable:=pTable, nElement:=0); *)
		pTmpTable	:= pTable + (SIZEOF(pTable^) * (UDINT#0));
		stElement1	:= pTmpTable^;
		(* ====================================================== *)
		IF stElement1.Position <> TableParameter.MinPosition THEN
			Error	:= TRUE;
			ErrorId	:= ERRORCODE_PARAMPOS;
			nState	:= 9999;
			RETURN;
		END_IF
		(* ====================================================== *)
		(* HKP: read table element with index (Parameter.nTableElements-1)	*)
		(* ====================================================== *)
		(* stElement1	:= F_GetCompensationElementAt(pTable:=pTable, nElement:=Parameter.nTableElements-1); *)
		pTmpTable	:= pTable + (SIZEOF(pTable^) * (TableParameter.NoOfTableElements-1));
		stElement1	:= pTmpTable^;
		(* ====================================================== *)
		IF stElement1.Position <> TableParameter.MaxPosition THEN
			Error	:= TRUE;
			ErrorId	:= ERRORCODE_PARAMPOS;
			nState	:= 9999;
			RETURN;
		END_IF
		(* HKP: This two parameter are not needed yet *)
		(* IF Parameter.eTableType <> TableType1DEquidistant OR Parameter.bModulo THEN
			Error	:= TRUE;
			ErrorId	:= ERRORCODE_TCNCNOTIMPL;
			nState	:= 9999;
			RETURN;
		END_IF *)

		(* check for equidistant table (table must contain in minimum 2 elements) *)
		pTmpTable	:= pTable + (SIZEOF(pTable^) * (UDINT#1));						(* read index 1 *)
		stElement2	:= pTmpTable^;
		pTmpTable	:= pTable + (SIZEOF(pTable^) * (UDINT#0));						(* read index 0 *)
		stElement1	:= pTmpTable^;
		fTmpDelta1	:= stElement2.Position - stElement1.Position;						(* calculate position delta 1: (index 1 - index 0) *)
		pTmpTable	:= pTable + (SIZEOF(pTable^) * (TableParameter.NoOfTableElements-1));	(* read index (n) *)
		stElement2	:= pTmpTable^;
		pTmpTable	:= pTable + (SIZEOF(pTable^) * (TableParameter.NoOfTableElements-2));	(* read index (n-1) *)
		stElement1	:= pTmpTable^;
		fTmpDelta2	:= stElement2.Position - stElement1.Position;						(* calculate position delta 2: (index (n) - index (n-1)) *)
		IF( ABS(fTmpDelta2 - fTmpDelta1) > 1.0E-6 ) THEN
			Error	:= TRUE;
			ErrorId	:= ERRORCODE_PARAMPOS;
			nState	:= 9999;
			RETURN;
		END_IF

		(* ====================================================== *)
		(* HKP: call action 'F_IsCompensationDirection()'				*)
		(* INPUT: eActive:=eActiveDirection, eRequested:=Parameter.Direction *)
		(* OUTPUT: bExecCalc									*)
		(* ====================================================== *)
		(* bExecCalc	:= F_IsCompensationDirection(eActive:=eActiveDirection, eRequested:=Parameter.Direction); *)
		ActIsCompensationDirection( );
		(* ====================================================== *)
		nState	:= 10;
	END_IF
10:
	(* ====================================================== *)
	(* HKP: call action 'F_IsCompensationDirection()'				*)
	(* INPUT: eActive:=eActiveDirection, eRequested:=Parameter.Direction *)
	(* OUTPUT: bExecCalc									*)
	(* ====================================================== *)
	(* bExecCalc	:= F_IsCompensationDirection(eActive:=eActiveDirection, eRequested:=Parameter.Direction); *)
	ActIsCompensationDirection( );
	(* ====================================================== *)
	IF NOT Enable THEN
		bExecCalc	:= FALSE;
		nState		:= 0;
	END_IF


9999:
	IF NOT Enable THEN
		nState	:= 0;
	END_IF

END_CASE


IF bExecCalc THEN
	(* compensation is generally enabled & direction is ok *)
	Active	:= TRUE;
	(* modulo or linear axis? *)
	IF( TableParameter.Modulo )THEN
		fSetPos	:= Axis.NcToPlc.ModuloSetPos;
	ELSE
		fSetPos	:= Axis.NcToPlc.SetPos;
	END_IF
	IF fSetPos < TableParameter.MinPosition THEN
		(* ====================================================== *)
		(* HKP: read table element with index (0)						*)
		(* ====================================================== *)
		(* stElement1	:= F_GetCompensationElementAt(pTable:=pTable, nElement:=0 ); *)
		pTmpTable	:= pTable + (SIZEOF(pTable^) * (UDINT#0));
		stElement1	:= pTmpTable^;
		(* ====================================================== *)
		Compensation	:= stElement1.Compensation;
	ELSIF fSetPos > TableParameter.MaxPosition THEN
		(* ====================================================== *)
		(* HKP: read table element with index (Parameter.nTableElements-1)	*)
		(* ====================================================== *)
		(* stElement1	:= F_GetCompensationElementAt(pTable:=pTable, nElement:=Parameter.nTableElements-1); *)
		pTmpTable	:= pTable + (SIZEOF(pTable^) * (TableParameter.NoOfTableElements-1));
		stElement1	:= pTmpTable^;
		(* ====================================================== *)
		Compensation := stElement1.Compensation;
	ELSE
		(* ====================================================== *)
		(* HKP: get left table index to position (Axis.NcToPlc.SetPos)		*)
		(* ====================================================== *)
		(* nLeftIndex	:= F_GetLeftIndex(fPos:=Axis.NcToPlc.SetPos, fMin:=Parameter.MinPosition, fMax:=Parameter.MaxPosition, nCount:=Parameter.NoOfTableElements); *)
		IF TableParameter.NoOfTableElements <= 1 THEN
			nLeftIndex := 0;
		ELSE
			IF fSetPos < TableParameter.MinPosition THEN
				nLeftIndex	:= 0;
			ELSIF fSetPos > TableParameter.MaxPosition THEN
				nLeftIndex	:= TableParameter.NoOfTableElements-1;
			ELSE
				fTmpStep	:= (TableParameter.MaxPosition-TableParameter.MinPosition)/UDINT_TO_LREAL(TableParameter.NoOfTableElements-1);
				nLeftIndex	:= LREAL_TO_UDINT(FLOOR((fSetPos-TableParameter.MinPosition)/fTmpStep));
			END_IF
		END_IF
		(* ====================================================== *)
		IF nLeftIndex >= TableParameter.NoOfTableElements-1 THEN
			(* there is no right index - probably fPos is exactly 'MaxPosition' *)
			(* ====================================================== *)
			(* HKP: read table element with index (Parameter.nTableElements-1)	*)
			(* ====================================================== *)
			(* stElement1	:= F_GetCompensationElementAt(pTable:=pTable, nElement:=Parameter.nTableElements-1); *)
			pTmpTable	:= pTable + (SIZEOF(pTable^) * (TableParameter.NoOfTableElements-1));
			stElement1	:= pTmpTable^;
			(* ====================================================== *)
			Compensation	:= stElement1.Compensation;
		ELSE
			(* ====================================================== *)
			(* HKP: read table element with index (nLeftIndex)				*)
			(* HKP: read table element with index (nLeftIndex+1)				*)
			(* ====================================================== *)
			(* stElement1	:= F_GetCompensationElementAt(pTable:=pTable, nElement:=nLeftIndex); *)
			(* stElement2	:= F_GetCompensationElementAt(pTable:=pTable, nElement:=nLeftIndex+1); *)
			pTmpTable	:= pTable + (SIZEOF(pTable^) * nLeftIndex);
			stElement1	:= pTmpTable^;
			pTmpTable	:= pTable + (SIZEOF(pTable^) * (nLeftIndex+1));
			stElement2	:= pTmpTable^;
			(* ====================================================== *)
			(* ====================================================== *)
			(* HKP: calculate linear interpolation between (stElement1) and (stElement2) for position (Axis.NcToPlc.SetPos)	*)
			(* ====================================================== *)
			(* Compensation	:= F_LinearInterpolationCompensation(fPos:=Axis.NcToPlc.SetPos, stElement1:=stElement1, stElement2:=stElement2); *)
			(* y := ax+b*)
			(* a:=(y2-y1)/(x2-x1)*)
			fTmpA	:= (stElement2.Compensation-stElement1.Compensation) / (stElement2.Position-stElement1.Position);
			(* b:=y-ax1 *)
			fTmpB	:= stElement1.Compensation - fTmpA*stElement1.Position;
			Compensation := fTmpA*fSetPos + fTmpB;
			(* ====================================================== *)
		END_IF
	END_IF
ELSE
	Compensation	:= 0.0;
	Active			:= FALSE;
END_IF
END_FUNCTION_BLOCK
ACTION ActIsCompensationDirection:
(*
FUNCTION F_IsCompensationDirection : BOOL
VAR_INPUT
	eActiveDirection		: E_WorkingDirection;	( eActive		: E_WorkingDirection )
	Parameter.Direction	: E_WorkingDirection;	( eRequested	: E_WorkingDirection )
END_VAR
VAR_OUTPUT
	bExecCalc		: BOOL;				( F_IsCompensationDirection : BOOL )
END_VAR
*)

(*
         |Active |       |       |       |
         |None   | both  | plus  | minus |
---------|-------|-------|-------|-------|
Req None |  0    |  0    |  0    |  0    |
---------|-------|-------|-------|-------|
Req both |  1    |  d.c. |  1    |  1    |
---------|-------|-------|-------|-------|
Req plus |  0    |  0    |  1    |  0    |
---------|-------|-------|-------|-------|
Req minus|  0    |  0    |  0    |  1    |
---------|-------|-------|-------|-------|

d.c.= don't care
*)

IF TableParameter.Direction = WorkDirectionBoth THEN
	bExecCalc	:= TRUE;
	RETURN;
END_IF
IF eActiveDirection = WorkDirectionPositive AND TableParameter.Direction = WorkDirectionPositive  THEN
	bExecCalc	:= TRUE;
	RETURN;
END_IF
IF eActiveDirection = WorkDirectionNegative AND TableParameter.Direction = WorkDirectionNegative  THEN
	bExecCalc	:= TRUE;
	RETURN;
END_IF
bExecCalc		:= FALSE;


(*
IF eActiveDirection = WorkingDirectionPlus AND (TableParameter.Direction = WorkingDirectionBoth OR TableParameter.Direction = WorkingDirectionPlus ) THEN
	bExecCalc	:= TRUE;
	RETURN;
END_IF
IF eActiveDirection = WorkingDirectionMinus AND (TableParameter.Direction = WorkingDirectionBoth OR TableParameter.Direction = WorkingDirectionMinus ) THEN
	bExecCalc	:= TRUE;
	RETURN;
END_IF
bExecCalc		:= FALSE;
*)
END_ACTION

(* POU _FB_ReadWriteParameter, ST *)
{library private}
FUNCTION_BLOCK _FB_ReadWriteParameter
VAR_IN_OUT
	Axis				:	AXIS_REF;
END_VAR
VAR_INPUT
	Enable			:	BOOL;
	ParameterNumber	:	MC_AxisParameter;
	Mode			:	INT; 		(* read/write *)
	ParameterType	:	INT;		(* bool/ not  bool *)
END_VAR
VAR_OUTPUT
	Done			:	BOOL;
	Busy: BOOL;
	Error			:	BOOL;
	ErrorID			:	UDINT;
	ADSbusy: BOOL;
END_VAR
VAR_IN_OUT
	ValueLreal		:	LREAL;
	ValueDword		:	DWORD;
	ValueBool		:	BOOL;
END_VAR
VAR
	iState			:	_E_TcMC_STATES := STATE_INITIALIZATION;
	fbAdsRead		:	ADSREAD;
	fbAdsWrite		:	ADSWRITE;

	dwValue			:	DWORD;
	lrValue			:	ARRAY[1..10] OF LREAL;
	NcBoolValue		:	UINT;

	bStarted			:	BOOL;
	stParaStruct		:	_ST_ParaStruct;
	n: INT;
	i: INT;
END_VAR
VAR CONSTANT
(*	ParaDWORD		:	INT:= 1;*)
	ParaLREAL		:	INT := 2;
(*	ParaBOOL		:	INT := 3;*)
END_VAR
(* ====================================================================== *)
(* *)
(* ====================================================================== *)

CASE iState OF
STATE_INITIALIZATION:	(* Ruhezustand *)
	Busy := FALSE;
    	IF Enable THEN
		(* initialize output values *)
		Done := FALSE;
		Error := FALSE;
		ErrorID := 0;

		stParaStruct.LrealSize := SIZEOF(lrValue[1]);
		stParaStruct.LrealOffset := 1;
		stParaStruct.Port := TcMcGlobal.NCPORT_TCMC; (* 2014-07-14 KSt *)

		(* some parameters are read immediately out of the cyclic axis interfaces *)
		(* other parameters are read via ADS, F_GetIndexGroup finds the required ADS parameters in this case *)
		IF Mode=READWRITEPARAMETERMODE_READ THEN
			CASE ParameterNumber OF
				CommandedPosition :
					stParaStruct.IndexOffset := 16#0000_0000;
					stParaStruct.IndexGroup := 0;
					stParaStruct.ParaType := ParaLreal;
					ValueLreal := Axis.NcToPlc.SetPos;
					Done := TRUE;
				ActualVelocity:
					stParaStruct.IndexOffset := 16#0000_0000;
					stParaStruct.IndexGroup := 0;
					stParaStruct.ParaType := ParaLreal;
					ValueLreal := Axis.NcToPlc.ActVelo;
					Done := TRUE;
				CommandedVelocity:
					stParaStruct.IndexOffset := 16#0000_0000;
					stParaStruct.IndexGroup := 0;
					stParaStruct.ParaType := ParaLreal;
					ValueLreal := Axis.NcToPlc.SetVelo;
					Done := TRUE;
				ELSE
					(* check index offset *)
					stParaStruct := _F_GetIndexGroup(ParaNumber := ParameterNumber, Mode:=Mode);
			END_CASE;
		ELSE
			(* check index offset *)
			stParaStruct := _F_GetIndexGroup(ParaNumber := ParameterNumber, Mode:=Mode);
		END_IF
		IF NOT Done THEN
			Busy := TRUE;
			iState := STATE_ORDER;
		END_IF
	ELSE
		Done := FALSE; (* reset with Enable=FALSE *)
		Error := FALSE;			(* reset at falling edge of Execute *)
		ErrorID := 0;
	END_IF
END_CASE

CASE iState OF
STATE_INITIALIZATION:
	;	(* already done before *)
STATE_ORDER :
		(* read via ADS *)
		IF FALSE AND (stParaStruct.ParaType <> ParameterType) (* no check !!*)
		THEN
			(* type mismatch *)
			Done := FALSE;
			ErrorID := MC_ERROR_COMMAND_NOT_ALLOWED;
			Error := TRUE;
		ELSIF stParaStruct.ParaType <> PARAMETERTYPE_NOTYPE THEN
			CASE Mode OF
(*------------------ Read parameter ---------------------------------------------------------------*)
				READWRITEPARAMETERMODE_READ	:
					IF stParaStruct.IndexGroup = 16#1000 (* no axis parameter *) AND
						(stParaStruct.IndexOffset=16#10 OR stParaStruct.IndexOffset=16#12) (* NC SAF or SVB cycle time *)
						THEN
						IF stParaStruct.ParaType=PARAMETERTYPE_DWORD THEN	(* read DWORD *)
								fbAdsRead(	NETID:= TcMcGlobal.NCNETID_TCMC,
(*									PORT:= TcMcGlobal.NCPORT_TCMC,*) (* 2014-07-14 KSt *)
									PORT:= stParaStruct.Port, (* 2014-07-14 KSt *)
									IDXGRP:= stParaStruct.IndexGroup,
									IDXOFFS:= stParaStruct.IndexOffset,
									LEN:= SIZEOF(dwValue),
									DESTADDR:= ADR(dwValue),
									READ:= TRUE,
									TMOUT:= TcMcGlobal.tADSTimeOut);
									ValueDword := 0;
									ValueLreal := DWORD_TO_LREAL(dwValue) * LREAL#100.0E-9;	(* convert to time value (SAF or SVB cycle time)*)
									ValueBool := 0;
						ELSE
							ErrorID := MC_ERROR_COMMAND_NOT_ALLOWED;
							Error := TRUE;
						END_IF

					ELSE (* axis data *)
						CASE stParaStruct.ParaType OF
							PARAMETERTYPE_DWORD :	(* read DWORD *)
								fbAdsRead(	NETID:= TcMcGlobal.NCNETID_TCMC,
(*									PORT:= TcMcGlobal.NCPORT_TCMC,*) (* 2014-07-14 KSt *)
									PORT:= stParaStruct.Port, (* 2014-07-14 KSt *)
									IDXGRP:= stParaStruct.IndexGroup+Axis.NcToPlc.AxisId,
									IDXOFFS:= stParaStruct.IndexOffset,
									LEN:= SIZEOF(dwValue),
									DESTADDR:= ADR(dwValue),
									READ:= TRUE,
									TMOUT:= TcMcGlobal.tADSTimeOut);
									ValueDword := dwValue; (* 20110511 KSt type conversion deleted for Tc3 *)
									ValueLreal := DWORD_TO_LREAL (dwValue);
									ValueBool := DWORD_TO_BOOL(dwValue);
								IF stParaStruct.IndexOffset=16#0000_0004 THEN
									ValueDword := 0;
									ValueLreal := DWORD_TO_LREAL(dwValue) * LREAL#1.0E-6;	(* convert to time value (axis cycle time)*)
									ValueBool := 0;
								END_IF
							PARAMETERTYPE_LREAL :		(* read LREAL *)
								fbAdsRead(	NETID:= TcMcGlobal.NCNETID_TCMC,
(*									PORT:= TcMcGlobal.NCPORT_TCMC,*) (* 2014-07-14 KSt *)
									PORT:= stParaStruct.Port, (* 2014-07-14 KSt *)
									IDXGRP:= stParaStruct.IndexGroup+Axis.NcToPlc.AxisId,
									IDXOFFS:= stParaStruct.IndexOffset,
									LEN:= MIN(SIZEOF(lrValue), stParaStruct.LrealSize),
									DESTADDR:= ADR(lrValue),
									READ:= TRUE,
									TMOUT:=  TcMcGlobal.tADSTimeOut);
									ValueLreal := lrValue[stParaStruct.LrealOffset];
									IF ValueLreal > 16#FFFF_FFFF THEN	(* 31.5.2007 KSt - avoid FPU exception *)
										ValueDword := 0;
										ValueBool := TRUE;
									ELSIF ValueLreal < -16#8000_0000 THEN 	(* 31.5.2007 KSt - avoid FPU exception *)
										ValueDword := 0;
										ValueBool := TRUE;
									ELSE
										ValueDword := LREAL_TO_DWORD(lrValue[stParaStruct.LrealOffset]); 	(* 31.5.2007 KSt - existing code *)
										ValueBool := LREAL_TO_BOOL(lrValue[stParaStruct.LrealOffset]);		(* 31.5.2007 KSt - existing code *)
									END_IF
	
							PARAMETERTYPE_BOOL :		(* read bool *)
								fbAdsRead(	NETID:= TcMcGlobal.NCNETID_TCMC,
(*									PORT:= TcMcGlobal.NCPORT_TCMC,*) (* 2014-07-14 KSt *)
									PORT:= stParaStruct.Port, (* 2014-07-14 KSt *)
									IDXGRP:= stParaStruct.IndexGroup+Axis.NcToPlc.AxisId,
									IDXOFFS:= stParaStruct.IndexOffset,
									LEN:= SIZEOF(NcBoolValue),
									DESTADDR:= ADR(NcBoolValue),
									READ:= TRUE,
									TMOUT:=  TcMcGlobal.tADSTimeOut);
									ValueBool := UINT_TO_BOOL(NcBoolValue);
									ValueDword := UINT_TO_DWORD(NcBoolValue);
									ValueLreal := UINT_TO_LREAL (NcBoolValue);
	
						END_CASE;
					END_IF
(*------------------ Write parameter ---------------------------------------------------------------*)
				READWRITEPARAMETERMODE_WRITE	:
					IF stParaStruct.IndexGroup = 16#1000 THEN (* no axis parameter *)
						ErrorID := MC_ERROR_COMMAND_NOT_ALLOWED;
						Error := TRUE;
					ELSE
						CASE stParaStruct.ParaType OF
							PARAMETERTYPE_DWORD:	(* read DWORD *)
								ValueDword := LREAL_TO_DWORD(ValueLreal);
								fbAdsWrite(	NETID:= TcMcGlobal.NCNETID_TCMC,
(*									PORT:= TcMcGlobal.NCPORT_TCMC,*) (* 2014-07-14 KSt *)
									PORT:= stParaStruct.Port, (* 2014-07-14 KSt *)
									IDXGRP:= stParaStruct.IndexGroup+Axis.NcToPlc.AxisId,
									IDXOFFS:= stParaStruct.IndexOffset,
									LEN:= SIZEOF(ValueDword),
									SRCADDR:= ADR(ValueDword),
									WRITE:= TRUE,
									TMOUT:= TcMcGlobal.tADSTimeOut);

							PARAMETERTYPE_LREAL :		(* read LREAL *)
								n := SIZEOF(lrValue) / SIZEOF(lrValue[1]);
								FOR i := 1 TO n DO lrValue[i] := 0; END_FOR
								lrValue[stParaStruct.LrealOffset] := ValueLreal;
								fbAdsWrite(	NETID:= TcMcGlobal.NCNETID_TCMC,
(*									PORT:= TcMcGlobal.NCPORT_TCMC,*) (* 2014-07-14 KSt *)
									PORT:= stParaStruct.Port, (* 2014-07-14 KSt *)
									IDXGRP:= stParaStruct.IndexGroup+Axis.NcToPlc.AxisId,
									IDXOFFS:= stParaStruct.IndexOffset,
									LEN:= MIN(SIZEOF(lrValue), stParaStruct.LrealSize),
									SRCADDR:= ADR(lrValue),
									WRITE:= TRUE,
									TMOUT:=  TcMcGlobal.tADSTimeOut);

							PARAMETERTYPE_BOOL :		(* read BOOL *)
								NcBoolValue := BOOL_TO_UINT(ValueBool);
								fbAdsWrite(	NETID:= TcMcGlobal.NCNETID_TCMC,
(*									PORT:= TcMcGlobal.NCPORT_TCMC,*) (* 2014-07-14 KSt *)
									PORT:= stParaStruct.Port, (* 2014-07-14 KSt *)
									IDXGRP:= stParaStruct.IndexGroup+Axis.NcToPlc.AxisId,
									IDXOFFS:= stParaStruct.IndexOffset,
									LEN:= SIZEOF(NcBoolValue),
									SRCADDR:= ADR(NcBoolValue),
									WRITE:= TRUE,
									TMOUT:=  TcMcGlobal.tADSTimeOut);
						END_CASE;
				END_IF
			END_CASE;

			bStarted := TRUE;
			CASE Mode OF
(*------------------ Read parameter ---------------------------------------------------------------*)
				READWRITEPARAMETERMODE_READ	:
					IF NOT fbAdsRead.Busy THEN
						bStarted := FALSE;
						iState := STATE_RUNNING;
					END_IF;
(*------------------ Write parameter ---------------------------------------------------------------*)
				READWRITEPARAMETERMODE_WRITE	:
					IF NOT fbAdsWrite.BUSY THEN
						bStarted := FALSE;
						iState := STATE_RUNNING;
					END_IF;
			END_CASE;
		ELSE
			Done := FALSE;
			ErrorID := MC_ERROR_COMMAND_NOT_ALLOWED;
			Error := TRUE;
			iState := STATE_INITIALIZATION;
		END_IF;

STATE_RUNNING:  (* wait *)
	IF NOT Error THEN
		CASE Mode OF
(*------------------ Read parameter ---------------------------------------------------------------*)
			READWRITEPARAMETERMODE_READ	:
				IF fbAdsRead.Err THEN
					ValueLreal := 0.0;
					ValueDword := 0;
					ValueBool := FALSE;
					Done := FALSE;
					ErrorID := fbAdsRead.ErrId;
					Error := TRUE;
					fbAdsRead(READ := FALSE);
					iState := STATE_INITIALIZATION;
				ELSE
					Done := TRUE;
					fbAdsRead(READ := FALSE);
			 		iState:=STATE_INITIALIZATION;
				END_IF;
(*------------------ Write parameter ---------------------------------------------------------------*)
			READWRITEPARAMETERMODE_WRITE	:
				IF fbAdsWrite.Err THEN
					Done := FALSE;
					ErrorID := fbAdsWrite.ErrId;
					Error := TRUE;
					fbAdsWrite(WRITE := FALSE);
					iState := STATE_INITIALIZATION;
				ELSE
					Done := TRUE;
					fbAdsWrite(WRITE := FALSE);
			 		iState:=STATE_INITIALIZATION;
				END_IF;
		END_CASE;
	ELSE
 		iState:=STATE_INITIALIZATION;
	END_IF;

ELSE  (* CASE : Unknown program state *)
	Error := TRUE;
	ErrorID := 16#FFFFFFFF;
	iState:=STATE_INITIALIZATION;
END_CASE;

ADSbusy := fbAdsWrite.BUSY OR fbAdsRead.BUSY;
IF iState=STATE_INITIALIZATION THEN
	(* reset Busy immediately  when sequence ends *)
	Busy := FALSE;
END_IF
END_FUNCTION_BLOCK

(* POU _FBAXIS_REF, ST *)
(*
	AXIS_REF data structure

	The FBAXIS_REF is actually not a function block but a data structure
	It includes the axis I/O variables as well as additional information.
	The reason for not using a STRUCT is that structures cannot hold
	located I/O variables.
	The user is supposed to use the AXIS_REF data type which internally
	redirects the type to this function block definition (alias).
*)
FUNCTION_BLOCK _FBAXIS_REF
VAR_INPUT
	PlcToNc 	AT %Q* 	: 	PLCTONC_AXIS_REF;
END_VAR
VAR_OUTPUT
	NcToPlc 	AT %I* 	:	NCTOPLC_AXIS_REF;
	ADS	 			: 	ST_AdsAddress;
	Status				:	ST_AxisStatus;
END_VAR
{library private}
VAR
	_internal : _InternalAxisRefData;
	Storage				:	ARRAY [0..127] OF DWORD;	(* universal storage for internal use *)
END_VAR
ReadStatus;
END_FUNCTION_BLOCK
ACTION ReadStatus:
(* NC cycle counter will be incremented after NC task updated the NcToPlc data structure *)
_internal.NcCycleCounter_AtReadStatusCall := SHR(NcToPlc.OpModeDWord, 24);

(* avoid multiple updates during one cycle which would cause additional CPU load *)
IF _internal.NcCycleCounter_AtReadStatusCall <> Status.NcCycleCounter OR _internal.NcCycleCounter_AtReadStatusCall=0 THEN

	(* new cycle - call status function *)
	_internal.LastTaskIndex_AtReadStatusCall := Status.UpdateTaskIndex;

	(* update the axis status
		ForceTaskIndexUpdate makes sure that the index of the current  task will be updated. 
		ForceTaskIndexUpdate=false saves time because a system call to gettaskindex will be avoided.
	*)
	Status := _F_ReadStatus( ForceTaskIndexUpdate:=_internal.CounterSameTaskIndex_AtReadStatusCall<100, NcToPlc := NcToPlc, PlcToNc := PlcToNc, LastStatus:=Status );

	(* count number of cycles with the same task index *)
	IF _internal.LastTaskIndex_AtReadStatusCall=Status.UpdateTaskIndex THEN
		IF _internal.CounterSameTaskIndex_AtReadStatusCall<100 THEN
			(* increment counter as long as the update task index does not change - max value is 100 *)
			_internal.CounterSameTaskIndex_AtReadStatusCall := _internal.CounterSameTaskIndex_AtReadStatusCall + 1;
		END_IF
	ELSE
		(* reset counter since update task index has changed - this is not supposed to happen but a user might call ReadStatus in several tasks *)
		_internal.CounterSameTaskIndex_AtReadStatusCall:= 0;
	END_IF
END_IF
END_ACTION

(* POU _MC_HaltPhasing, FBD *)
FUNCTION_BLOCK _MC_HaltPhasing
VAR_IN_OUT
	Master 			: 	AXIS_REF;
	Slave 			: 	AXIS_REF;
END_VAR
VAR_INPUT
	Execute			:	BOOL;	(* B *)	(* Start the motion at rising edge *)
	Deceleration		:	LREAL;	(* E *)	(* Value of the maximum deceleration *)
	Jerk				:	LREAL;	(* E *)	(* Value of the maximum jerk *)
	BufferMode		:	MC_BufferMode;		(* E *)
	Options			: 	ST_PhasingOptions;	(* V *)	(* optional parameters *)
END_VAR
VAR_OUTPUT
	Done			:	BOOL;	(* B *)
	Busy			: 	BOOL;	(* E *)
	Active			: 	BOOL;	(* E *)
	CommandAborted	:	BOOL;	(* E *)
	Error			:	BOOL;	(* B *)
	ErrorID			:	UDINT;	(* E *)
END_VAR
VAR
	PhasingGeneric : _FB_PhasingGeneric;
END_VAR
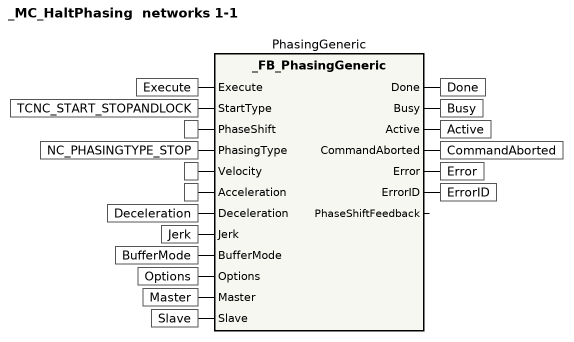
_FBD_ (* Function Block Diagram *)
NETWORK 1
	PhasingGeneric:_FB_PhasingGeneric(Execute: Execute, StartType: TCNC_START_STOPANDLOCK, PhaseShift: , PhasingType: NC_PHASINGTYPE_STOP, Velocity: , Acceleration: , Deceleration: Deceleration, Jerk: Jerk, BufferMode: BufferMode, Options: Options, Master: Master, Slave: Slave, Busy => Busy, Active => Active, CommandAborted => CommandAborted, Error => Error, ErrorID => ErrorID) => Done
_END_FBD_
END_FUNCTION_BLOCK

(* POU _MC_PhasingAbsolute, FBD *)
FUNCTION_BLOCK _MC_PhasingAbsolute
(*
	This Function Block creates an absolute phase shift in the master position of a slave axis. 
	The master position is shifted in relation to the real physical position. This is analogous 
	to opening a coupling on the master shaft for a moment, and is used to delay or advance 
	an axis to its master. The phase shift is seen from the slave. The master does not know 
	that there is a phase shift experienced by the slave (MasterPos as seen from the 
	SlaveAxis = PhysicalMasterPos + PhaseShiftValueSlaveAxis, the phase shift value has 
	the character of a position offset) The phase shift remains until another ‘Phasing’ 
	command changes it again.
*)
VAR_IN_OUT
	Master 			: 	AXIS_REF;
	Slave 			: 	AXIS_REF;
END_VAR
VAR_INPUT
	Execute			:	BOOL;	(* B *)	(* Start the motion at rising edge *)
	PhaseShift		:	LREAL;	(* B *)	(* Target position for the motion *)
	Velocity			:	LREAL;	(* E *)	(* Value of the maximum velocity *)
	Acceleration		:	LREAL;	(* E *)	(* Value of the maximum acceleration *)
	Deceleration		:	LREAL;	(* E *)	(* Value of the maximum deceleration *)
	Jerk				:	LREAL;	(* E *)	(* Value of the maximum jerk *)
	BufferMode		:	MC_BufferMode;		(* E *)
	Options			: 	ST_PhasingOptions;	(* V *)	(* optional parameters *)
END_VAR
VAR_OUTPUT
	Done			:	BOOL;	(* B *)
	Busy			: 	BOOL;	(* E *)
	Active			: 	BOOL;	(* E *)
	CommandAborted	:	BOOL;	(* E *)
	Error			:	BOOL;	(* B *)
	ErrorID			:	UDINT;	(* E *)
	AbsolutePhaseShift : 	LREAL;	(* E *)
END_VAR
VAR
	PhasingGeneric : _FB_PhasingGeneric;
END_VAR
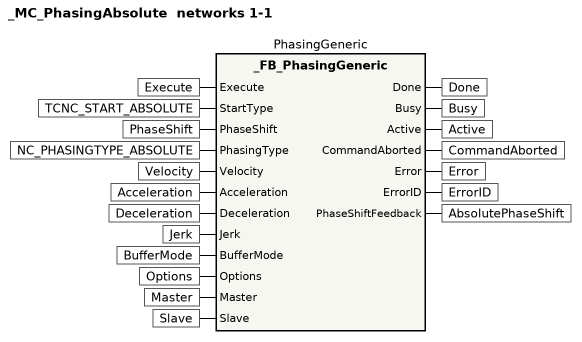
_FBD_ (* Function Block Diagram *)
NETWORK 1
	PhasingGeneric:_FB_PhasingGeneric(Execute: Execute, StartType: TCNC_START_ABSOLUTE, PhaseShift: PhaseShift, PhasingType: NC_PHASINGTYPE_ABSOLUTE, Velocity: Velocity, Acceleration: Acceleration, Deceleration: Deceleration, Jerk: Jerk, BufferMode: BufferMode, Options: Options, Master: Master, Slave: Slave, Busy => Busy, Active => Active, CommandAborted => CommandAborted, Error => Error, ErrorID => ErrorID, PhaseShiftFeedback => AbsolutePhaseShift) => Done
_END_FBD_
(* the same logic as Structured Text *)
(* Network 1 *)
PhasingGeneric(Execute := Execute, StartType := TCNC_START_ABSOLUTE, PhaseShift := PhaseShift, PhasingType := NC_PHASINGTYPE_ABSOLUTE, Velocity := Velocity, Acceleration := Acceleration, Deceleration := Deceleration, Jerk := Jerk, BufferMode := BufferMode, Options := Options, Master := Master, Slave := Slave);
Busy := PhasingGeneric.Busy;
Active := PhasingGeneric.Active;
CommandAborted := PhasingGeneric.CommandAborted;
Error := PhasingGeneric.Error;
ErrorID := PhasingGeneric.ErrorID;
AbsolutePhaseShift := PhasingGeneric.PhaseShiftFeedback;
Done := PhasingGeneric.Done;
END_FUNCTION_BLOCK

(* POU _MC_PhasingRelative, FBD *)
FUNCTION_BLOCK _MC_PhasingRelative
(*
	This Function Block creates a phase shift in the master position of a slave axis relative 
	to the existing phase shift.
	The master position is shifted in relation to the real physical position. This is analogous 
	to opening a coupling on the master shaft for a moment, and is used to delay or advance 
	an axis to its master. The phase shift is seen from the slave. The master does not know 
	that there is a phase shift experienced by the slave. (MasterPos as seen from 
	SlaveAxis = PhysicalMasterPos + PhaseShiftValueSlaveAxis, the phase shift value has 
	the character of a position offset) The phase shift remains until another ‘Phasing’ 
	command changes it again. Relative phase shifts are added to each other for the 
	applicable phase shift
*)
VAR_IN_OUT
	Master 			: 	AXIS_REF;
	Slave 			: 	AXIS_REF;
END_VAR
VAR_INPUT
	Execute			:	BOOL;	(* B *)	(* Start the motion at rising edge *)
	PhaseShift		:	LREAL;	(* B *)	(* Target position for the motion *)
	Velocity			:	LREAL;	(* E *)	(* Value of the maximum velocity *)
	Acceleration		:	LREAL;	(* E *)	(* Value of the maximum acceleration *)
	Deceleration		:	LREAL;	(* E *)	(* Value of the maximum deceleration *)
	Jerk				:	LREAL;	(* E *)	(* Value of the maximum jerk *)
	BufferMode		:	MC_BufferMode;		(* E *)
	Options			: 	ST_PhasingOptions;	(* V *)	(* optional parameters *)
END_VAR
VAR_OUTPUT
	Done			:	BOOL;	(* B *)
	Busy			: 	BOOL;	(* E *)
	Active			: 	BOOL;	(* E *)
	CommandAborted	:	BOOL;	(* E *)
	Error			:	BOOL;	(* B *)
	ErrorID			:	UDINT;	(* E *)
	CoveredPhaseShift : 	LREAL;	(* E *)
END_VAR
VAR
	PhasingGeneric : _FB_PhasingGeneric;
END_VAR
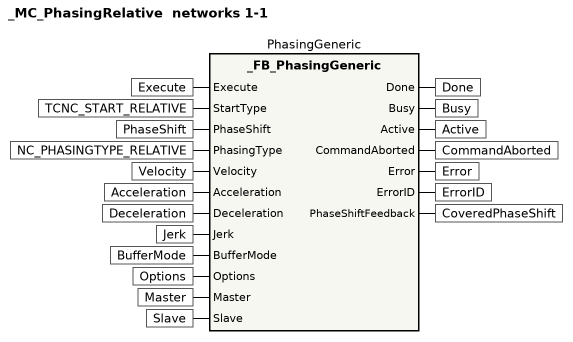
_FBD_ (* Function Block Diagram *)
NETWORK 1
	PhasingGeneric:_FB_PhasingGeneric(Execute: Execute, StartType: TCNC_START_RELATIVE, PhaseShift: PhaseShift, PhasingType: NC_PHASINGTYPE_RELATIVE, Velocity: Velocity, Acceleration: Acceleration, Deceleration: Deceleration, Jerk: Jerk, BufferMode: BufferMode, Options: Options, Master: Master, Slave: Slave, Busy => Busy, Active => Active, CommandAborted => CommandAborted, Error => Error, ErrorID => ErrorID, PhaseShiftFeedback => CoveredPhaseShift) => Done
_END_FBD_
(* the same logic as Structured Text *)
(* Network 1 *)
PhasingGeneric(Execute := Execute, StartType := TCNC_START_RELATIVE, PhaseShift := PhaseShift, PhasingType := NC_PHASINGTYPE_RELATIVE, Velocity := Velocity, Acceleration := Acceleration, Deceleration := Deceleration, Jerk := Jerk, BufferMode := BufferMode, Options := Options, Master := Master, Slave := Slave);
Busy := PhasingGeneric.Busy;
Active := PhasingGeneric.Active;
CommandAborted := PhasingGeneric.CommandAborted;
Error := PhasingGeneric.Error;
ErrorID := PhasingGeneric.ErrorID;
CoveredPhaseShift := PhasingGeneric.PhaseShiftFeedback;
Done := PhasingGeneric.Done;
END_FUNCTION_BLOCK

(* POU _TcMC_ADSRDWRT, ST *)
FUNCTION_BLOCK _TcMC_ADSRDWRT (* Extended ADS read/write command *)
(*
 	This function block substitutes the generic ADSRDWRT/EX command.
	This block waits for an update of the cyclic NcToPlc interface after 
	the ADS command has been successfully executed.
*)
VAR_IN_OUT
	Axis 			: 	AXIS_REF;
END_VAR
VAR_INPUT
	NETID			:	T_AmsNetId;
	PORT			:	T_AmsPort;
	IDXGRP			:	UDINT;
	IDXOFFS		:	UDINT;
	WRITELEN		:	UDINT;
	READLEN		:	UDINT;
	SRCADDR 		:	DWORD;
	DESTADDR 		:	DWORD;
	WRTRD			:	BOOL;
	TMOUT			:	TIME := DEFAULT_ADS_TIMEOUT;
END_VAR
VAR_OUTPUT
	BUSY			:	BOOL;
	ERR			:	BOOL;
	ERRID			:	UDINT;
	COUNT_R		:	UDINT;				(* count of bytes actually read *)
END_VAR
VAR
	fbAdsRdWrt				: 	FW_AdsRdWrt;
	NcCycleCounter			: 	BYTE;
	NcCycleCounterAdsEnd	: 	BYTE;
	UpdateCounter			:	BYTE;
	NoUpdateCounter 		: 	BYTE;	(* used for timeout detection *)
	state: INT;
END_VAR
CASE state OF
 0 :	(* call ADS *)
	fbAdsRdWrt(
		sNetId := NETID,
		nPort := PORT,
		nIdxGrp := IDXGRP,
		nIdxOffs := IDXOFFS,
		cbWriteLen := WRITELEN,
		cbReadLen := READLEN,
		pWriteBuff := SRCADDR,
		pReadBuff := DESTADDR,
		bExecute := WRTRD,
		tTimeout := TMOUT
		);
	IF fbAdsRdWrt.bBusy THEN
		BUSY := TRUE;
		ERR := FALSE;
		ERRID := 0;
		COUNT_R := 0;
		UpdateCounter:=0;
		NoUpdateCounter:=0;
		state := state + 1;
	END_IF

 1 :	(* wait till ADS call is finished *)
	fbAdsRdWrt();
	IF NOT fbAdsRdWrt.bBusy THEN
		IF fbAdsRdWrt.bError THEN
			(* error - feedback without any delay *)
			BUSY := FALSE;
			ERR := fbAdsRdWrt.bError;
			ERRID := fbAdsRdWrt.nErrId;
			COUNT_R := fbAdsRdWrt.cbRead;
			fbAdsRdWrt(bExecute := WRTRD);
			state := 0;
		ELSE
			(* save current NC cycle counter to check for AXIS_REF update in the next state *)
			NcCycleCounter := _F_UpdateNcCycleCounter(Axis);(* store cycle counter at the end of the ADS command sequence *)
			NcCycleCounterAdsEnd := NcCycleCounter;
			state := state + 1;
		END_IF
	END_IF

 2 :	(* wait for AXIS_REF update *)
	IF _F_NcCycleCounterUpdated( LastNcCycleCounter:=NcCycleCounter, Axis:=Axis ) THEN
		UpdateCounter := UpdateCounter + 1;
	ELSE
		NoUpdateCounter:=NoUpdateCounter+1;
		IF NoUpdateCounter>100 THEN
			BUSY := FALSE;
			ERR := TRUE;
			ERRID := MC_ERROR_NCCYCLECOUNTERUPDATE;
			fbAdsRdWrt(bExecute := WRTRD);
			state := 0;
		END_IF
	END_IF
	NcCycleCounter := _F_UpdateNcCycleCounter(Axis);(* store cycle counter when leaving this command *)

	IF UpdateCounter >= 2 THEN	(* at least two updates after response on ADS command *)
		BUSY := FALSE;
		ERR := fbAdsRdWrt.bError;
		ERRID := fbAdsRdWrt.nErrId;
		COUNT_R := fbAdsRdWrt.cbRead;
		fbAdsRdWrt(bExecute := WRTRD);
		state := 0;
	END_IF
END_CASE
END_FUNCTION_BLOCK

(* POU _TcMC_ADSREAD, ST *)
FUNCTION_BLOCK _TcMC_ADSREAD (* Extended ADS read command *)
(*
 	This function block substitutes the generic ADSREAD/EX command.
	This block waits for an update of the cyclic NcToPlc interface after 
	the ADS command has been successfully executed.
*)
VAR_IN_OUT
	Axis 			: 	AXIS_REF;
END_VAR
VAR_INPUT
	NETID			:	T_AmsNetId;
	PORT			:	T_AmsPort;
	IDXGRP			:	UDINT;
	IDXOFFS		:	UDINT;
	LEN				:	UDINT;
	DESTADDR 		:	DWORD;
	READ			:	BOOL;
	TMOUT			:	TIME := DEFAULT_ADS_TIMEOUT;
END_VAR
VAR_OUTPUT
	BUSY			:	BOOL;
	ERR			:	BOOL;
	ERRID			:	UDINT;
	COUNT_R		:	UDINT;	(* count of bytes actually read *)
END_VAR
VAR
	fbAdsRead				: 	FW_AdsRead;
	NcCycleCounter			: 	BYTE;
	NcCycleCounterAdsEnd	: 	BYTE;
	UpdateCounter			:	BYTE;
	NoUpdateCounter 		: 	BYTE;	(* used for timeout detection *)
	state: INT;
END_VAR
CASE state OF
 0 :	(* call ADS *)
	fbAdsRead(
		sNetId := NETID,
		nPort := PORT,
		nIdxGrp := IDXGRP,
		nIdxOffs := IDXOFFS,
		cbReadLen := LEN,
		pReadBuff := DESTADDR,
		bExecute := READ,
		tTimeout := TMOUT
		);
	IF fbAdsRead.bBusy THEN
		BUSY := TRUE;
		ERR := FALSE;
		ERRID := 0;
		COUNT_R := 0;
		UpdateCounter:=0;
		NoUpdateCounter:=0;
		state := state + 1;
	END_IF

 1 :	(* wait till ADS call is finished *)
	fbAdsRead();
	IF NOT fbAdsRead.bBusy THEN
		IF fbAdsRead.bError THEN
			(* error - feedback without any delay *)
			BUSY := FALSE;
			ERR := fbAdsRead.bError;
			ERRID := fbAdsRead.nErrId;
			COUNT_R := fbAdsRead.cbRead;
			fbAdsRead(bExecute := READ);
			state := 0;
		ELSE
			(* save current NC cycle counter to check for AXIS_REF update in the next state *)
			NcCycleCounter := _F_UpdateNcCycleCounter(Axis);(* store cycle counter at the end of the ADS command sequence *)
			NcCycleCounterAdsEnd := NcCycleCounter;
			state := state + 1;
		END_IF
	END_IF

 2 :	(* wait for AXIS_REF update *)
	IF _F_NcCycleCounterUpdated( LastNcCycleCounter:=NcCycleCounter, Axis:=Axis ) THEN
		UpdateCounter := UpdateCounter + 1;
	ELSE
		NoUpdateCounter:=NoUpdateCounter+1;
		IF NoUpdateCounter>100 THEN
			BUSY := FALSE;
			ERR := TRUE;
			ERRID := MC_ERROR_NCCYCLECOUNTERUPDATE;
			fbAdsRead(bExecute := READ);
			state := 0;
		END_IF
	END_IF
	NcCycleCounter := _F_UpdateNcCycleCounter(Axis);(* store cycle counter when leaving this command *)

	IF UpdateCounter >= 2 THEN	(* at least two updates after response on ADS command *)
		BUSY := FALSE;
		ERR := fbAdsRead.bError;
		ERRID := fbAdsRead.nErrId;
		COUNT_R := fbAdsRead.cbRead;
		fbAdsRead(bExecute := READ);
		state := 0;
	END_IF
END_CASE
END_FUNCTION_BLOCK

(* POU _TcMC_ADSWRITE, ST *)
FUNCTION_BLOCK _TcMC_ADSWRITE (* ADS write command *)
(*
 	This function block substitutes the generic ADSWRITE command.
	This block waits for an update of the cyclic NcToPlc interface after 
	the ADS command has been successfully executed.
*)
VAR_IN_OUT
	Axis 			: 	AXIS_REF;
END_VAR
VAR_INPUT
	NETID			:	T_AmsNetId;
	PORT			:	T_AmsPort;
	IDXGRP			:	UDINT;
	IDXOFFS		:	UDINT;
	LEN				:	UDINT;
	SRCADDR 		:	DWORD;
	WRITE			:	BOOL;
	TMOUT			:	TIME := DEFAULT_ADS_TIMEOUT;
END_VAR
VAR_OUTPUT
	BUSY			:	BOOL;
	ERR			:	BOOL;
	ERRID			:	UDINT;
END_VAR
VAR
	fbAdsWrite				: 	FW_AdsWrite;
	NcCycleCounter			: 	BYTE;
	NcCycleCounterAdsEnd	: 	BYTE;
	UpdateCounter			:	BYTE;
	NoUpdateCounter 		: 	BYTE;	(* used for timeout detection *)
	state: INT;
END_VAR
CASE state OF
 0 :	(* call ADS *)
	fbAdsWrite(
		sNetId := NETID,
		nPort := PORT,
		nIdxGrp := IDXGRP,
		nIdxOffs := IDXOFFS,
		cbWriteLen := LEN,
		pWriteBuff := SRCADDR,
		bExecute := WRITE,
		tTimeout := TMOUT
		);
	IF fbAdsWrite.bBusy THEN
		BUSY := TRUE;
		ERR := FALSE;
		ERRID := 0;
		UpdateCounter:=0;
		NoUpdateCounter:=0;
		state := state + 1;
	END_IF

 1 :	(* wait till ADS call is finished *)
	fbAdsWrite();
	IF NOT fbAdsWrite.bBusy THEN
		IF fbAdsWrite.bError THEN
			(* error - feedback without any delay *)
			BUSY := FALSE;
			ERR := fbAdsWrite.bError;
			ERRID := fbAdsWrite.nErrId;
			fbAdsWrite(bExecute := WRITE);
			state := 0;
		ELSE
			(* save current NC cycle counter to check for AXIS_REF update in the next state *)
			NcCycleCounter := _F_UpdateNcCycleCounter(Axis);(* store cycle counter at the end of the ADS command sequence *)
			NcCycleCounterAdsEnd := NcCycleCounter;
			state := state + 1;
		END_IF
	END_IF

 2 :	(* wait for AXIS_REF update *)
	IF _F_NcCycleCounterUpdated( LastNcCycleCounter:=NcCycleCounter, Axis:=Axis ) THEN
		UpdateCounter := UpdateCounter + 1;
	ELSE
		NoUpdateCounter:=NoUpdateCounter+1;
		IF NoUpdateCounter>100 THEN
			BUSY := FALSE;
			ERR := TRUE;
			ERRID := MC_ERROR_NCCYCLECOUNTERUPDATE;
			fbAdsWrite(bExecute := WRITE);
			state := 0;
		END_IF
	END_IF
	NcCycleCounter := _F_UpdateNcCycleCounter(Axis);(* store cycle counter when leaving this command *)

	IF UpdateCounter >= 2 THEN	(* at least two updates after response on ADS command *)
		BUSY := FALSE;
		ERR := fbAdsWrite.bError;
		ERRID := fbAdsWrite.nErrId;
		fbAdsWrite(bExecute := WRITE);
		state := 0;
	END_IF
END_CASE
END_FUNCTION_BLOCK

(* POU _TCMCGLOBAL, ST *)
(*	Global constants and parameters *)
FUNCTION_BLOCK _TCMCGLOBAL
VAR_INPUT
	NCPORT_TCMC 				:	UINT 	:= AMSPORT_R0_NC;  (* 20110511 type changed from INT to UINT *)
	NCPORT_TCMC_COUPLING	:	UINT 	:= AMSPORT_R0_NC; (* used with all axis coupling commands - 12.7.2006 KSt *)  (* 20110511 type changed from INT to UINT *)
	NCNETID_TCMC 				:	T_AmsNetId := '';
	NCPORT_TCMC_CAM 		:	UINT 	:= AMSPORT_R0_NC; (* 20110511 type changed from INT to UINT *)
	NCNETID_TCMC_CAM		:	T_AmsNetId := '';
	NCPORT_TCMC_SUPERPOSITION	:	UINT 	:= AMSPORT_R0_NCSAF; (* 20140930 KSt added *)
END_VAR
VAR_OUTPUT
	NcDeviceInfoTcMainVersion 	: 	DWORD;
	NcDeviceInfoTcSubVersion 	: 	DWORD;
	NcDeviceInfoNcDriverVersion 	: 	DWORD;
	NcDeviceInfoNcVersion		: 	DWORD;
	NcDeviceInfoNcName			: 	STRING(19);
END_VAR
VAR CONSTANT
	Axis 	: _ST_NCADS_Axis;	(* IDXGRP and IDXOFFS constants of axis parameter/status/functions *)
	Table 	: _ST_NCADS_Table;	(* IDXGRP and IDXOFFS constants of table parameter/status/functions *)

	NCPORT_TCNCCAMMING_TABLEFUNCTION	: 	UINT	:=	500;

	(* timeout *)
	tTargetPosTimeOut			:	TIME	:= T#6s; (* 20050128 KSt - changed from 5 sec to 6 sec to be later than a NC PEH error (5 sec) *)
	tADSTimeOut   				:	TIME	:= T#1s;
	tStopMonitoringTimeOut		:	TIME	:= T#100ms;	(* 20111208 KSt - new for stop monitoring (axis in standstill window *)

	NCTOPLC_FEEDBACK_MAXWAITCYCLES : INT := 10; (* maximum number of PLC cycles to wait for a cyclic feedback in NcToPlc after an ADS command *)
END_VAR
VAR
	fbADSRDDEVINFO: ADSRDDEVINFO;
	DeviceVersion: DWORD;
END_VAR
;
END_FUNCTION_BLOCK
ACTION ReadDeviceInfo:
(* get current NC version *)
(* this piece of code will be executed just once *)
IF  DeviceVersion = 0 THEN
	IF fbADSRDDEVINFO.ERR THEN
		fbADSRDDEVINFO( RDINFO:= FALSE );
		fbADSRDDEVINFO( RDINFO:= TRUE );
	END_IF

	fbADSRDDEVINFO(
		NETID:= '',
		PORT:= 500,
		RDINFO:= TRUE,
		TMOUT:= T#1s,
		DEVNAME=> NcDeviceInfoNcName,
		DEVVER=> DeviceVersion);

	NcDeviceInfoTcMainVersion := DeviceVersion AND 16#FF;;
	NcDeviceInfoTcSubVersion := (DeviceVersion / 16#100) AND 16#FF;
	NcDeviceInfoNcDriverVersion :=(DeviceVersion / 16#10000) AND 16#FFFF;
	NcDeviceInfoNcVersion := NcDeviceInfoTcMainVersion * 16#1000000 + NcDeviceInfoTcSubVersion * 16#10000 + NcDeviceInfoNcDriverVersion;
END_IF
END_ACTION

(* POU F_AxisCamDataQueued, ST *)
FUNCTION F_AxisCamDataQueued : BOOL
(* 	reference: 	NC -> PLC axis interface (128 bytes)
	check if bit 22 of an axis StateDWord is set:
	New cam data has been queued to a slave axis which is coupled to master via a cam table. 
	The flag comes up when the PLC modifies the camming data.
	Das Flag wird TRUE, wenn neue bzw. veränderte Kurvenscheibendaten von der SPS an 
	eine Slave-Achse gesendet werden.
*)
VAR_INPUT
	StateDWord : DWORD;
END_VAR
VAR
END_VAR
F_AxisCamDataQueued := (StateDWord AND 2#0000_0000_0100_0000_0000_0000_0000_0000) <> 0;
END_FUNCTION

(* POU F_AxisCamScalingPending, ST *)
FUNCTION F_AxisCamScalingPending : BOOL
(* 	reference: 	NC -> PLC axis interface (128 bytes)
	check if bit 23 of an axis StateDWord is set:
	- The flag signals that the scaling and/or offset setting of a cam table has been requested 
	to be performed 	at a certain master position. This request is pending while the function 
	result is TRUE and has been executed after a falling edge of this signal.
	- Das Flag zeigt an das die Skalierung und/oder das Setzen der Offsets einer Kurvenscheibe
	beauftrag wurde aber erst später (ab einer bestimmten Master-Position) durchgeführt wird.
	Mit fallender Flanke des Signals wurde der Auftrag ausgeführt.
*)
VAR_INPUT
	StateDWord : DWORD;
END_VAR
VAR
END_VAR
F_AxisCamScalingPending := (StateDWord AND 2#0000_0000_1000_0000_0000_0000_0000_0000) <> 0;
END_FUNCTION

(* POU F_AxisCamTableQueued, ST *)
FUNCTION F_AxisCamTableQueued : BOOL
(* 	reference: 	NC -> PLC axis interface (128 bytes)
	check if bit 21 of an axis StateDWord is set:
	New cam data has been queued to a slave axis which is coupled to master via a cam table. 
	The flag comes up when the PLC modifies the camming data.
	Das Flag wird TRUE, wenn neue bzw. veränderte Kurvenscheibendaten von der SPS an 
	eine Slave-Achse gesendet werden.
*)
VAR_INPUT
	StateDWord : DWORD;
END_VAR
VAR
END_VAR
F_AxisCamTableQueued := (StateDWord AND 2#0000_0000_0010_0000_0000_0000_0000_0000) <> 0;
END_FUNCTION

(* POU F_AxisExternalLatchValid, ST *)
FUNCTION F_AxisExternalLatchValid : BOOL
(* 	reference: 	NC -> PLC axis interface (128 bytes)
	check if bit 16 of an axis StateDWord is set:
	External latch value or sensing switch has become valid
	Externer Latchwert bzw. Messtaster gültig geworden
*)
VAR_INPUT
	StateDWord : DWORD;
END_VAR
VAR
END_VAR
F_AxisExternalLatchValid := (StateDWord AND 2#0000_0000_0000_0001_0000_0000_0000_0000) <> 0;
END_FUNCTION

(* POU F_AxisGotNewTargetPosition, ST *)
FUNCTION F_AxisGotNewTargetPosition  : BOOL
(* 	reference: 	NC -> PLC axis interface (128 bytes)
	check if bit 17 of an axis StateDWord is set:
	Axis got a new target position or a new velocity
	while the current move command is in execution.
	Die Zielposition oder die Geschwindigkeit der Achse
	wurde geändert, während die Achse eine Bewegung ausführt
*)
VAR_INPUT
	StateDWord : DWORD;
END_VAR
VAR
END_VAR
F_AxisGotNewTargetPosition := (StateDWord AND 2#0000_0000_0000_0010_0000_0000_0000_0000) <> 0;
END_FUNCTION

(* POU F_AxisInPTPmode, ST *)
FUNCTION F_AxisInPTPmode : BOOL
(* 	reference: 	NC -> PLC axis interface (128 bytes)
	check if bit 25 of an axis StateDWord is set:
	- The flag signals that the axis accepts PTP motion commands. That requires that the axis is 
	not coupled to other axes and not part of a NC-I or FIFO group.
	- Das Flag zeigt an, dass die Achse PTP Bewegungskommandos entgegen nimmt. Das setzt 
	voraus, dass die Achse nicht gekoppelt ist oder in eine NC-I oder FIFO-Gruppe integriert ist.
*)
VAR_INPUT
	StateDWord : DWORD;
END_VAR
VAR
END_VAR
F_AxisInPTPmode := (StateDWord AND 2#0000_0010_0000_0000_0000_0000_0000_0000) <> 0;
END_FUNCTION

(* POU F_AxisIoDataIsInvalid, ST *)
FUNCTION F_AxisIoDataIsInvalid : BOOL
(* 	reference: 	NC -> PLC axis interface (128 bytes)
	check if bit 30 of an axis StateDWord is set:
	Axis I/O data is invalid  (e.g. invalid 'WcState' or 'CdlState' )
	Achse hat keine gültigen I/O-Daten  (e.g. invalid 'WcState' or 'CdlState' )
*)
VAR_INPUT
	StateDWord : DWORD;
END_VAR
VAR
END_VAR
F_AxisIoDataIsInvalid := (StateDWord AND 2#0100_0000_0000_0000_0000_0000_0000_0000) <> 0;
END_FUNCTION

(* POU F_AxisIsCalibrated, ST *)
FUNCTION F_AxisIsCalibrated : BOOL
(* 	reference: 	NC -> PLC axis interface (128 bytes)
	check if bit 1 of an axis StateDWord is set:
	Axis has been referenced ("Axis calibrated")
	Achse ist referenziert ("Achse geeicht")
*)
VAR_INPUT
	StateDWord : DWORD;
END_VAR
VAR
END_VAR
F_AxisIsCalibrated := (StateDWord AND 2#0000_0000_0000_0000_0000_0000_0000_0010) <> 0;
END_FUNCTION

(* POU F_AxisIsMoving, ST *)
FUNCTION F_AxisIsMoving : BOOL
(* 	reference: 	NC -> PLC axis interface (128 bytes)
	check if bit 9 OR 10 of an axis StateDWord is set:
	Axis moving (forward or backwards)
	Achse fährt (vorwärts oder rückwärts)
*)
VAR_INPUT
	StateDWord : DWORD;
END_VAR
VAR
END_VAR
F_AxisIsMoving := (StateDWord AND 2#0000_0000_0000_0000_0000_0110_0000_0000) <> 0;
END_FUNCTION

(* POU F_AxisIsMovingBackwards, ST *)
FUNCTION F_AxisIsMovingBackwards : BOOL
(* 	reference: 	NC -> PLC axis interface (128 bytes)
	check if bit 10 of an axis StateDWord is set:
	Axis moving to logically smaller values
	Achse fährt logisch kleiner
*)
VAR_INPUT
	StateDWord : DWORD;
END_VAR
VAR
END_VAR
F_AxisIsMovingBackwards := (StateDWord AND 2#0000_0000_0000_0000_0000_0100_0000_0000) <> 0;
END_FUNCTION

(* POU F_AxisIsMovingForward, ST *)
FUNCTION F_AxisIsMovingForward : BOOL
(* 	reference: 	NC -> PLC axis interface (128 bytes)
	check if bit 9 of an axis StateDWord is set:
	Axis moving to logically larger values
	Achse fährt logisch größer
*)
VAR_INPUT
	StateDWord : DWORD;
END_VAR
VAR
END_VAR
F_AxisIsMovingForward := (StateDWord AND 2#0000_0000_0000_0000_0000_0010_0000_0000) <> 0;
END_FUNCTION

(* POU F_AxisIsNotMoving, ST *)
FUNCTION F_AxisIsNotMoving : BOOL
(* 	reference: 	NC -> PLC axis interface (128 bytes)
	check if bit 2 of an axis StateDWord is set:
	Axis is logically stationary ("Axis not moving")
	Achse ist im logischen Stillstand ("Achse fährt nicht")
*)
VAR_INPUT
	StateDWord : DWORD;
END_VAR
VAR
END_VAR
F_AxisIsNotMoving := (StateDWord AND 2#0000_0000_0000_0000_0000_0000_0000_0100) <> 0;
END_FUNCTION

(* POU F_AxisIsReady, ST *)
FUNCTION F_AxisIsReady : BOOL
(* 	reference: 	NC -> PLC axis interface (128 bytes)
	check if bit 0 of an axis StateDWord is set:
	Axis is ready for operation
	Achse ist betriebsbereit
*)
VAR_INPUT
	StateDWord : DWORD;
END_VAR
VAR
END_VAR
F_AxisIsReady := (StateDWord AND 2#0000_0000_0000_0000_0000_0000_0000_0001) <> 0;
END_FUNCTION

(* POU F_AxisJobPending, ST *)
FUNCTION F_AxisJobPending : BOOL
(* 	reference: 	NC -> PLC axis interface (128 bytes)
	check if bit 24 of an axis StateDWord is set:
	- The flag signals that the a new motion job ist pending and will be 
	   executed after the active job is finished (buffer mode)
	- Das Flag zeigt an das die ein neuer Fahrauftrag gepuffert ist,
	   um nach dem aktuellen Auftrag ausgeführt zu werden (buffer mode)
*)
VAR_INPUT
	StateDWord : DWORD;
END_VAR
VAR
END_VAR
F_AxisJobPending := (StateDWord AND 2#0000_0001_0000_0000_0000_0000_0000_0000) <> 0;
END_FUNCTION

(* POU F_GetVersion_TcMC2, ST *)
FUNCTION F_GetVersion_TcMC2 : UINT	(* Gets the library version info *)
VAR_INPUT
	nVersionElement		:	INT;
END_VAR
(*
	Possible nVersionElement parameter:
	1	:	major number
	2	:	minor number
	3	:	revision number
*)

